febInvalidCallUpdownPatternNo(CLK:= bCallPB AND bInvalidCallUpdownPatternNoHold  , Q=> );

IF febInvalidCallUpdownPatternNo.Q THEN
bInvalidCallUpdownPatternNoPulse := TRUE;
END_IF

tInvalidCallUpdownPatternNoPulseTimer(IN:=bInvalidCallUpdownPatternNoPulse , PT:=t#0.5s , Q=> , ET=> );

IF tInvalidCallUpdownPatternNoPulseTimer.Q OR NOT bCallPB THEN
bInvalidCallUpdownPatternNoPulse := FALSE;
END_IF

IF bCallPBRE.Q AND NOT bInvalidCallUpdownPatternNoHold THEN
bCallCompleted := FALSE;
CallStep:= 1;
END_IF


CASE CallStep OF

1:

Call_DSUpdownPattern := ARDsUpdownPatternMemory[Call_iUpDownPatternNo];

CallStep := 11;


10:
bCallCompleted := TRUE;
CallSelfCheckHR := FALSE;
PreviousUpdownPatternCallNo := Call_iUpDownPatternNo;
CallStep := 99;

11:

bCallCompleted := TRUE;
CallStep := 99;



99:
;
END_CASE

END_FUNCTION_BLOCK

// ---- FBs/B_JKS_NewFB/FBP-Memory_Sub/fbA31_ArmSpeedProfileMemory.TcPOU
FUNCTION_BLOCK fbA31_ArmSpeedProfileMemory

VAR_INPUT
	bSavePB : BOOL;
	bLoadPB : BOOL;
	bCopyPB : BOOL;
	iCopyToSpdProfileNo : INT;
	iVertMaxVelo : INT;
	iVertMaxAcc : INT;
	iVertMaxDcc : INT;
	iVertMinVelo : INT;
	iVertMinAcc : INT;
	iVertMinDcc : INT;
END_VAR


VAR_IN_OUT PERSISTENT

	iArmSpdProfileNo: INT; (* 10 sets of Station Sequence Recipe *)
	DSArmSpeedProfile : DSA31_ArmSpeedProfileMemory;

	Call_iArmSpdProfile : INT;
	bCallPB: BOOL;

END_VAR
VAR_OUTPUT
	bSaveInd: BOOL;
	bLoadInd: BOOL;
	bCallCompleted : BOOL;
	bInvalidCallArmSpdProfileNoHold: BOOL;
	bInvalidCallArmSpdProfileNoPulse: BOOL;
	Call_DSArmSpeedProfile : DSA31_ArmSpeedProfileMemory;

END_VAR
VAR
	SaveIndHr: BOOL;
	LoadIndHr: BOOL;

	SaveTimerDelay: TON;
	LoadTimerDelay: TON;
	SelfCheckTimer: TON;
	bLoadEn: BOOL;
	SelfCheckloopArmSpdProfileRecipe: BOOL;
	PreviousArmSpdProfileRecipe: INT;

	LoadDF : R_TRIG;
	LoadENDF : R_TRIG;

	SaveDF: R_TRIG;
	CallIntervalTimer: TON;
	CallIntervalDIFU: R_TRIG;

	bCallCompletedHR: BOOL;
	bCallCompletedHRRE: R_TRIG;
	CallCompletedTimer: TON;
	CallSelfCheckTimer : TON;
	CallSelfCheckloop : BOOL;

	CallSelfCheckRE: R_TRIG;
	CallStep: INT;
	CallSelfCheckHR: BOOL;
	bCallPBRE: R_TRIG;

	LoadFL: INT;
	SaveFL: INT;
	PreviousArmSpdProfileCallNo: INT;
	CallSFL: INT;
	febInvalidCallArmSpdProfileNo: F_TRIG;



	rebInvalidCallArmSpdProfileNo: R_TRIG;
	tInvalidCallArmSpdProfileNoPulseTimer: TON;
	CopyDF: R_TRIG;
	iMaxMinFL: INT;
END_VAR

VAR PERSISTENT

	ARDsArmSpeedProfileMemory : ARRAY [1..iArmSpeedProfileArrayQty] OF DSA31_ArmSpeedProfileMemory;
	ARsStorageArmSpeedProfileDescription: ARRAY [0..iArmSpeedProfileArrayQty] OF STRING(50);


END_VAR

IF iArmSpdProfileNo < 1 THEN
iArmSpdProfileNo := 1;
END_IF

IF iArmSpdProfileNo > iArmSpeedProfileArrayQty THEN
iArmSpdProfileNo := iArmSpeedProfileArrayQty;
END_IF



(*Min / Max Control*)
			IF DSArmSpeedProfile.lrSpeedVelo < iVertMinVelo THEN
			DSArmSpeedProfile.lrSpeedVelo:= iVertMinVelo;
			ELSIF DSArmSpeedProfile.lrSpeedVelo > iVertMaxVelo THEN
			DSArmSpeedProfile.lrSpeedVelo:= iVertMaxVelo;
			END_IF

			IF DSArmSpeedProfile.lrAcc < iVertMinAcc THEN
			DSArmSpeedProfile.lrAcc:= iVertMinAcc;
			ELSIF DSArmSpeedProfile.lrAcc > iVertMaxAcc THEN
			DSArmSpeedProfile.lrAcc:= iVertMaxAcc;
			END_IF

			IF DSArmSpeedProfile.lrDcc < iVertMinDcc THEN
			DSArmSpeedProfile.lrDcc:= iVertMinDcc;
			ELSIF DSArmSpeedProfile.lrDcc > iVertMaxDcc THEN
			DSArmSpeedProfile.lrDcc:= iVertMaxDcc;
			END_IF



(*Load and Save Indicator*)
IF bSavePB THEN
SaveIndHr := TRUE;
END_IF

SaveTimerDelay(IN:=SaveIndHr, PT := T#1s, Q=>, ET=>);
IF SaveTimerDelay.Q THEN
SaveIndHr := FALSE;
END_IF

IF SaveIndHr AND NOT SaveTimerDelay.Q THEN
bSaveInd := TRUE;
ELSE
bSaveInd := FALSE;
END_IF

IF bLoadPB THEN
LoadIndHr := TRUE;
END_IF

LoadTimerDelay(IN:=LoadIndHr, PT := T#1s, Q=>, ET=>);
IF loadtimerdelay.Q THEN
LoadIndHr := FALSE;
END_IF

IF loadIndHr AND NOT LoadTimerDelay.Q THEN
bLoadInd := TRUE;
ELSE
bLoadInd := FALSE;
END_IF

IF iArmSpdProfileNo <> PreviousArmSpdProfileRecipe THEN
bLoadEn := TRUE;
ELSE
bLoadEn := FALSE;
END_IF


(* Load Recipe *)

LoadDF(CLK:=bLoadPB,Q=>);
LoadENDF(CLK:=bLoadEn,Q=>);

IF LoadDF.Q OR LoadENDF.Q THEN

DSArmSpeedProfile := ARDsArmSpeedProfileMemory[iArmSpdProfileNo];
PreviousArmSpdProfileRecipe := iArmSpdProfileNo  ;

END_IF


(* Save Recipe *)

SaveDF(CLK:=bSavePB,Q=>);

IF SaveDF.Q THEN

ARDsArmSpeedProfileMemory[iArmSpdProfileNo] := DSArmSpeedProfile;
ARsStorageArmSpeedProfileDescription[iArmSpdProfileNo] := DSArmSpeedProfile.sDescription;

END_IF


(*Copy Recipe*)

CopyDF(CLK:=bCopyPB,Q=>);

IF CopyDF.Q THEN

ARDsArmSpeedProfileMemory[iCopyToSpdProfileNo] := ARDsArmSpeedProfileMemory[iArmSpdProfileNo];
ARsStorageArmSpeedProfileDescription[iCopyToSpdProfileNo] := ARDsArmSpeedProfileMemory[iArmSpdProfileNo].sDescription;

END_IF





(* Call Recipe *)
(* ---- Call Recipe Complete Flag ---*)


IF NOT bCallPB THEN
bCallCompleted := FALSE;
END_IF

bCallPBRE(CLK:=bCallPB , Q=> );

IF (Call_iArmSpdProfile <= 0 OR Call_iArmSpdProfile > iArmSpeedProfileArrayQty) AND bCallPB THEN
bInvalidCallArmSpdProfileNoHold := TRUE;
ELSE
bInvalidCallArmSpdProfileNoHold := FALSE;
END_IF


febInvalidCallArmSpdProfileNo(CLK:= bCallPB AND bInvalidCallArmSpdProfileNoHold  , Q=> );

IF febInvalidCallArmSpdProfileNo.Q THEN
bInvalidCallArmSpdProfileNoPulse := TRUE;
END_IF

tInvalidCallArmSpdProfileNoPulseTimer(IN:=bInvalidCallArmSpdProfileNoPulse , PT:=t#0.5s , Q=> , ET=> );

IF tInvalidCallArmSpdProfileNoPulseTimer.Q OR NOT bCallPB THEN
bInvalidCallArmSpdProfileNoPulse := FALSE;
END_IF

IF bCallPBRE.Q AND NOT bInvalidCallArmSpdProfileNoHold THEN
bCallCompleted := FALSE;
CallStep:= 1;
END_IF


CASE CallStep OF

1:

Call_DSArmSpeedProfile := ARDsArmSpeedProfileMemory[Call_iArmSpdProfile];

CallStep := 11;


10:
bCallCompleted := TRUE;
CallSelfCheckHR := FALSE;
PreviousArmSpdProfileCallNo := Call_iArmSpdProfile;
CallStep := 99;

11:

bCallCompleted := TRUE;
CallStep := 99;



99:
;
END_CASE

END_FUNCTION_BLOCK

// ---- FBs/B_JKS_NewFB_V2/FBP-Memory_Sub/fbV2_A32_MachineZoneHeight.TcPOU
FUNCTION_BLOCK fbV2_A32_MachineZoneHeight

VAR_IN_OUT PERSISTENT

	ARDSLdZoneHeight : ARRAY [0..iLdStnQty] OF DSA32_StationZoneHeight;
	ARDSStationZoneHeight : ARRAY [0..iStnQty] OF DSA32_StationZoneHeight;
	ARDSUldZoneHeight : ARRAY [0..iUldStnQty] OF DSA32_StationZoneHeight;


END_VAR
VAR_OUTPUT
	ARDSLdZonePosOut : ARRAY [0..iLdStnQty] OF DSA32_StationZonePosOut;
	ARDSStationZonePosOut : ARRAY [0..iStnQty] OF DSA32_StationZonePosOut;
	ARDSUldZonePosOut : ARRAY [0..iUldStnQty] OF DSA32_StationZonePosOut;

END_VAR
VAR PERSISTENT

	ARfbLdStationZoneHeight : ARRAY [0..iLdStnQty] OF fbA32_StationZoneHeight;
	ARfbStationZoneHeight : ARRAY [0..iStnQty] OF fbA32_StationZoneHeight;
	ARfbUldStationZoneHeight : ARRAY [0..iUldStnQty] OF fbA32_StationZoneHeight;

END_VAR
VAR
	Loop: INT;
END_VAR

(*Loading*)

Loop := 1;
IF Loop >= 1 THEN
	FOR Loop := 1 TO iLdStnQty DO
		(*Loading*)
		IF Loop >= 1 AND Loop <= iLdStnQty THEN
		ARfbLdStationZoneHeight[Loop](DSStationZoneHeight:=ARDSLdZoneHeight[Loop] , DSStationZonePosOut=>ARDSLdZonePosOut[Loop] );
		END_IF
	END_FOR
END_IF

Loop := 1;
IF Loop >= 1 THEN
	FOR Loop := 1 TO iStnQty DO
		(*Station Qty*)
		IF Loop >= 1 AND Loop <= iStnQty THEN
		ARfbStationZoneHeight[Loop](DSStationZoneHeight:=ARDSStationZoneHeight[Loop] , DSStationZonePosOut=>ARDSStationZonePosOut[Loop] );
		END_IF
	END_FOR
END_IF

Loop := 1;
IF Loop >= 1 THEN
	FOR Loop := 1 TO iUldStnQty DO
		(*Unloading*)
		IF Loop >= 1 AND Loop <= iUldStnQty THEN
		ARfbUldStationZoneHeight[Loop](DSStationZoneHeight:=ARDSUldZoneHeight[Loop] , DSStationZonePosOut=>ARDSUldZonePosOut[Loop] );
		END_IF
	END_FOR
END_IF

END_FUNCTION_BLOCK

// ---- FBs/B_JKS_NewFB/FBP-Memory_Sub/fbA32_StationZoneHeight.TcPOU
FUNCTION_BLOCK fbA32_StationZoneHeight
VAR_IN_OUT PERSISTENT

	DSStationZoneHeight : DSA32_StationZoneHeight;


END_VAR
VAR_OUTPUT
	DSStationZonePosOut : DSA32_StationZonePosOut;

END_VAR
VAR
	bZone1RangeValid: BOOL;
	bZone2RangeValid: BOOL;
	bZone3RangeValid: BOOL;
	bZone4RangeValid: BOOL;
END_VAR

DSStationZonePosOut.lrZone1StartPos := DSStationZoneHeight.lrTopPos;
DSStationZonePosOut.lrZone2StartPos := DSStationZonePosOut.lrZone1EndPos;
DSStationZonePosOut.lrZone3StartPos := DSStationZonePosOut.lrZone2EndPos;
DSStationZonePosOut.lrZone4StartPos := DSStationZonePosOut.lrZone3EndPos;

DSStationZonePosOut.lrZone1EndPos := DSStationZoneHeight.lrTopPos + DSStationZoneHeight.lrZone1Range;
DSStationZonePosOut.lrZone2EndPos := DSStationZoneHeight.lrTopPos + DSStationZoneHeight.lrZone1Range + DSStationZoneHeight.lrZone2Range;
DSStationZonePosOut.lrZone3EndPos := DSStationZoneHeight.lrTopPos + DSStationZoneHeight.lrZone1Range + DSStationZoneHeight.lrZone2Range + DSStationZoneHeight.lrZone3Range;
DSStationZonePosOut.lrZone4EndPos := DSStationZoneHeight.lrBottomPos;

DSStationZonePosOut.lrMidPos := DSStationZoneHeight.lrMidPos; (*Added New*)

DSStationZoneHeight.lrZone4Range := DSStationZoneHeight.lrBottomPos - DSStationZonePosOut.lrZone3EndPos;

IF DSStationZoneHeight.lrZone1Range > (DSStationZoneHeight.lrBottomPos - DSStationZoneHeight.lrTopPos) THEN
DSStationZoneHeight.lrZone1Range := DSStationZoneHeight.lrBottomPos - DSStationZoneHeight.lrTopPos;
END_IF

IF DSStationZoneHeight.lrZone2Range > (DSStationZoneHeight.lrBottomPos - DSStationZoneHeight.lrZone1Range - DSStationZoneHeight.lrTopPos) THEN
DSStationZoneHeight.lrZone2Range := DSStationZoneHeight.lrBottomPos - DSStationZoneHeight.lrZone1Range - DSStationZoneHeight.lrTopPos;
END_IF

IF DSStationZoneHeight.lrZone3Range > (DSStationZoneHeight.lrBottomPos - DSStationZoneHeight.lrZone1Range - DSStationZoneHeight.lrZone2Range - DSStationZoneHeight.lrTopPos) THEN
DSStationZoneHeight.lrZone3Range := DSStationZoneHeight.lrBottomPos - DSStationZoneHeight.lrZone1Range - DSStationZoneHeight.lrZone2Range - DSStationZoneHeight.lrTopPos;
END_IF


IF DSStationZoneHeight.lrZone1Range < 0 THEN
DSStationZoneHeight.lrZone1Range := 0;
ELSIF DSStationZoneHeight.lrZone2Range < 0 THEN
DSStationZoneHeight.lrZone2Range := 0;
ELSIF DSStationZoneHeight.lrZone3Range < 0 THEN
DSStationZoneHeight.lrZone3Range := 0;
END_IF







IF DSStationZoneHeight.lrZone1Range <> 0 THEN
bZone1RangeValid := TRUE;
ELSE
bZone1RangeValid := FALSE;
END_IF

IF DSStationZoneHeight.lrZone2Range <> 0 THEN
bZone2RangeValid := TRUE;
ELSE
bZone2RangeValid := FALSE;
END_IF

IF DSStationZoneHeight.lrZone3Range <> 0 THEN
bZone3RangeValid := TRUE;
ELSE
bZone3RangeValid := FALSE;
END_IF

IF DSStationZoneHeight.lrZone4Range <> 0 THEN
bZone4RangeValid := TRUE;
ELSE
bZone4RangeValid := FALSE;
END_IF

END_FUNCTION_BLOCK

// ---- POUs/MainProgram/AutoArmCtrl/PosConfirmBitCtrl_Arm1.TcPOU
PROGRAM PosConfirmBitCtrl_Arm1
VAR

	fbFBPArmHorzZoneConfirm_Arm1 : fbV2_FBPArmHorzZoneConfirm;

END_VAR

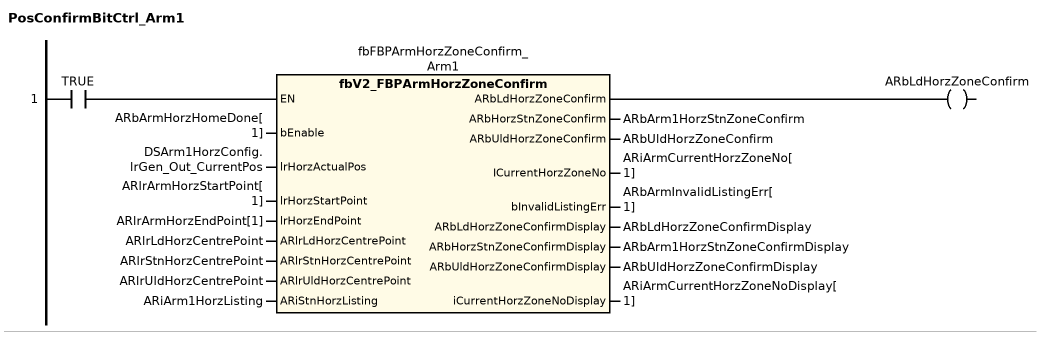
// NETWORK 1
fbFBPArmHorzZoneConfirm_Arm1(
    bEnable := ARbArmHorzHomeDone[1],
    lrHorzActualPos := DSArm1HorzConfig.lrGen_Out_CurrentPos,
    lrHorzStartPoint := ARlrArmHorzStartPoint[1],
    lrHorzEndPoint := ARlrArmHorzEndPoint[1],
    ARlrLdHorzCentrePoint := ARlrLdHorzCentrePoint,
    ARlrStnHorzCentrePoint := ARlrStnHorzCentrePoint,
    ARlrUldHorzCentrePoint := ARlrUldHorzCentrePoint,
    ARiStnHorzListing := ARiArm1HorzListing,
    ARbHorzStnZoneConfirm => ARbArm1HorzStnZoneConfirm,
    ARbUldHorzZoneConfirm => ARbUldHorzZoneConfirm,
    ICurrentHorzZoneNo => ARiArmCurrentHorzZoneNo[1],
    bInvalidListingErr => ARbArmInvalidListingErr[1],
    ARbLdHorzZoneConfirmDisplay => ARbLdHorzZoneConfirmDisplay,
    ARbHorzStnZoneConfirmDisplay => ARbArm1HorzStnZoneConfirmDisplay,
    ARbUldHorzZoneConfirmDisplay => ARbUldHorzZoneConfirmDisplay,
    iCurrentHorzZoneNoDisplay => ARiArmCurrentHorzZoneNoDisplay[1]); // fbV2_FBPArmHorzZoneConfirm
ARbLdHorzZoneConfirm := fbFBPArmHorzZoneConfirm_Arm1.ARbLdHorzZoneConfirm;

END_PROGRAM

// ---- FBs/B_JKS_NewFB_V2/FBP-ArmRelated/fbV2_FBPArmHorzZoneConfirm.TcPOU
FUNCTION_BLOCK fbV2_FBPArmHorzZoneConfirm
VAR_INPUT
	bEnable 					: BOOL;
(*	ARiLdStnID					: INT;
	ARiUldStnID					: INT;
*)	lrHorzActualPos 			: LREAL;
	lrHorzStartPoint 			: LREAL;
	lrHorzEndPoint 			: LREAL;
	ARlrLdHorzCentrePoint 	: ARRAY [0..iLdStnQty] OF LREAL;
	ARlrStnHorzCentrePoint 	: ARRAY [0..iStnQty] OF LREAL;
	ARlrUldHorzCentrePoint 	: ARRAY [0..iUldStnQty] OF LREAL;
	ARiStnHorzListing 		: ARRAY [1..50] OF INT;

END_VAR


VAR_OUTPUT
	ARbLdHorzZoneConfirm 		: ARRAY [0..iLdStnQty] OF BOOL;
	ARbHorzStnZoneConfirm 		: ARRAY [1..iStnQty] OF BOOL;
	ARbUldHorzZoneConfirm 		: ARRAY [0..iUldStnQty] OF BOOL;
	ICurrentHorzZoneNo 			: INT;
	bInvalidListingErr				: BOOL;

	ARbLdHorzZoneConfirmDisplay 		: ARRAY [0..iLdStnQty] OF BOOL;
	ARbHorzStnZoneConfirmDisplay 	: ARRAY [1..iStnQty] OF BOOL;
	ARbUldHorzZoneConfirmDisplay 	: ARRAY [0..iUldStnQty] OF BOOL;
	iCurrentHorzZoneNoDisplay 		: INT;

END_VAR
(*
VAR_IN_OUT
	iZoneEndPoint : ARRAY [1..20] OF INT;
	iActualPos: INT;

END_VAR
*)
VAR

	iActualPos: INT;


	bEnableRE: R_TRIG;
	iGenZoneFL: INT;
	ARlrZoneCentrePoint : ARRAY [1..50] OF LREAL;
	ARlrZoneEndPoint : ARRAY [1..50] OF LREAL;
	ARbZonePosConfirmInt : ARRAY [1..50] OF BOOL;
	iCheckListFL: INT;
	iEndPointFL: INT;
	bEnableFE: F_TRIG;
	iClearFL: INT;
	IZonePosCfFL: INT;
	iCurrentStnFL: INT;
	bCheckStnConfirm: BOOL;
	iCheckStnBitFL: INT;
	iGenZoneSFL: INT;
	bStnHorzListingFound: BOOL;
	bCurrentHorzZoneNoFound: BOOL;
END_VAR

(*bEnable Rising Edge*)
bEnableRE(CLK:=bEnable , Q=> );
bEnableFE(CLK:=bEnable , Q=> );


(*Generate Zone Centre Point and Transfer Confirm Bit*)
IF bEnable THEN
iGenZoneFL := 1;
	FOR iGenZoneFL := 1 TO 50 DO
		IF iGenZoneFL >= 1 AND iGenZoneFL <= 50 THEN

		bStnHorzListingFound := FALSE;

			iGenZoneSFL := 1;
				FOR iGenZoneSFL := 1 TO iLdStnQty DO
					IF iGenZoneSFL >= 1 AND iGenZoneSFL <= iLdStnQty THEN

						IF ARiStnHorzListing[iGenZoneFL] = ARiLdStnID[iGenZoneSFL] THEN
							ARlrZoneCentrePoint[iGenZoneFL] := ARlrLdHorzCentrePoint[iGenZoneSFL];
							ARbLdHorzZoneConfirm[iGenZoneSFL] := ARbZonePosConfirmInt[iGenZoneFL];
							bStnHorzListingFound := TRUE;
						END_IF

					END_IF
				END_FOR

			iGenZoneSFL := 1;
				FOR iGenZoneSFL := 1 TO iUldStnQty DO
					IF iGenZoneSFL >= 1 AND iGenZoneSFL <= iUldStnQty THEN

						IF ARiStnHorzListing[iGenZoneFL] = ARiUldStnID[iGenZoneSFL] THEN
							ARlrZoneCentrePoint[iGenZoneFL] := ARlrUldHorzCentrePoint[iGenZoneSFL];
							ARbUldHorzZoneConfirm[iGenZoneSFL] := ARbZonePosConfirmInt[iGenZoneFL];
							bStnHorzListingFound := TRUE;
						END_IF

					END_IF
				END_FOR


			IF NOT bStnHorzListingFound (*ARiStnHorzListing[iGenZoneFL] <> ARiUldStnID AND ARiStnHorzListing[iGenZoneFL] <> ARiUldStnID*) AND ARiStnHorzListing[iGenZoneFL] <> 0 AND ARiStnHorzListing[iGenZoneFL] <= iStnQty THEN
				ARlrZoneCentrePoint[iGenZoneFL] := ARlrStnHorzCentrePoint[ARiStnHorzListing[iGenZoneFL]];
				ARbHorzStnZoneConfirm[ARiStnHorzListing[iGenZoneFL]] := ARbZonePosConfirmInt[iGenZoneFL];
			END_IF


		END_IF
	END_FOR
END_IF


(*Check invalid Stn Listing*)
IF bEnableRE.Q THEN
bInvalidListingErr := FALSE;
iCheckListFL := 1;
	FOR iCheckListFL := 1 TO 50 DO
		IF iCheckListFL >= 1 AND iCheckListFL <= 50 THEN

			IF iCheckListFL = 1 AND ARlrZoneCentrePoint[1] <= 0 THEN
			bInvalidListingErr := TRUE;
			iCheckListFL := 50+1;
			END_IF

			IF iCheckListFL > 1 AND ARlrZoneCentrePoint[iCheckListFL] <= ARlrZoneCentrePoint[iCheckListFL-1] AND ARiStnHorzListing[iCheckListFL] >0 THEN
			bInvalidListingErr := TRUE;
			iCheckListFL := 50+1;
			END_IF
		END_IF
	END_FOR
END_IF




(*Generate End Point *)
IF bEnableRE.Q THEN
iEndPointFL := 1;
	FOR iEndPointFL := 1 TO 50 DO
		IF iEndPointFL >= 1 AND iEndPointFL <= 50-1 THEN

(*			IF iEndPointFL >1 THEN*)
				IF ((ARlrZoneCentrePoint[iEndPointFL+1] - ARlrZoneCentrePoint[iEndPointFL])/2) >0 THEN
				ARlrZoneEndPoint[iEndPointFL] := ((ARlrZoneCentrePoint[iEndPointFL+1] - ARlrZoneCentrePoint[iEndPointFL])/2)+ARlrZoneCentrePoint[iEndPointFL];
				ELSIF lrHorzEndPoint <= ARlrZoneCentrePoint[iEndPointFL] THEN
				ARlrZoneEndPoint[iEndPointFL] := ARlrZoneCentrePoint[iEndPointFL]+5000;
				iEndPointFL := 50+1;
				ELSIF lrHorzEndPoint > ARlrZoneCentrePoint[iEndPointFL] THEN
				ARlrZoneEndPoint[iEndPointFL] := lrHorzEndPoint+1;
				iEndPointFL := 50+1;
				END_IF
(*			END_IF*)
		END_IF
	END_FOR
END_IF


(*Clear Data*)
IF bEnableFE.Q THEN
iClearFL := 1;
	FOR iClearFL := 1 TO 50 DO
		IF iClearFL >= 1 AND iClearFL <= 50 THEN

			ARlrZoneCentrePoint[iClearFL] := 0;
			ARlrZoneEndPoint[iClearFL] := 0;
			ARbZonePosConfirmInt[iClearFL] := FALSE;

			IF iClearFL >= 1 AND iClearFL <= iStnQty THEN
			ARbHorzStnZoneConfirm[iClearFL] := FALSE;
			END_IF

			IF iClearFL >= 1 AND iClearFL <= iLdStnQty THEN
			ARbLdHorzZoneConfirm[iClearFL] := FALSE;
			END_IF

			IF iClearFL >= 1 AND iClearFL <= iUldStnQty THEN
			ARbUldHorzZoneConfirm[iClearFL] := FALSE;
			END_IF

		END_IF
	END_FOR



ICurrentHorzZoneNo := 0;
bInvalidListingErr := FALSE;
END_IF


(*Convert LREAL to INT*)


iActualPos := LREAL_TO_INT(lrHorzActualPos);




IF bEnable AND NOT bInvalidListingErr THEN


(*General Zone Pos Confirm Internal*)
IZonePosCfFL := 1;
	FOR IZonePosCfFL := 1 TO 50 DO
		IF IZonePosCfFL >= 1 AND IZonePosCfFL <= 50 THEN

			IF IZonePosCfFL = 1 THEN
				IF (iActualPos >= lrHorzStartPoint) AND (iActualPos < ARlrZoneEndPoint[IZonePosCfFL]) AND iActualPos >0 THEN
				ARbZonePosConfirmInt[IZonePosCfFL] := TRUE;
				ELSE
				ARbZonePosConfirmInt[IZonePosCfFL] := FALSE;
				END_IF
			END_IF

			IF IZonePosCfFL > 1 THEN
				IF (iActualPos >= ARlrZoneEndPoint[IZonePosCfFL-1]) AND (iActualPos < ARlrZoneEndPoint[IZonePosCfFL]) AND iActualPos >0 THEN
				ARbZonePosConfirmInt[IZonePosCfFL] := TRUE;
				ELSE
				ARbZonePosConfirmInt[IZonePosCfFL] := FALSE;
				END_IF
			END_IF
		END_IF
	END_FOR

(*Generate ICurrentHorzZoneNo *)
	bCurrentHorzZoneNoFound := FALSE;


		IF NOT bCurrentHorzZoneNoFound THEN

		iCurrentStnFL := 1;
			FOR iCurrentStnFL := 1 TO iLdStnQty DO
				IF iCurrentStnFL >= 1 AND iCurrentStnFL <= iLdStnQty THEN

					IF ARbLdHorzZoneConfirm[iCurrentStnFL] THEN
					ICurrentHorzZoneNo := ARiLdStnID[iCurrentStnFL];
					bCurrentHorzZoneNoFound := TRUE;
					END_IF

				END_IF
			END_FOR
		END_IF


		IF NOT bCurrentHorzZoneNoFound THEN

		iCurrentStnFL := 1;
			FOR iCurrentStnFL := 1 TO iUldStnQty DO
				IF iCurrentStnFL >= 1 AND iCurrentStnFL <= iUldStnQty THEN

					IF ARbUldHorzZoneConfirm[iCurrentStnFL] THEN
					ICurrentHorzZoneNo := ARiUldStnID[iCurrentStnFL];
					bCurrentHorzZoneNoFound := TRUE;
					END_IF

				END_IF
			END_FOR
		END_IF

		IF NOT bCurrentHorzZoneNoFound THEN

		iCurrentStnFL := 1;
			FOR iCurrentStnFL := 1 TO iStnQty DO
				IF iCurrentStnFL >= 1 AND iCurrentStnFL <= iStnQty THEN

					IF ARbHorzStnZoneConfirm[iCurrentStnFL] THEN
					ICurrentHorzZoneNo := iCurrentStnFL;
					bCurrentHorzZoneNoFound := TRUE;
					END_IF

				END_IF
			END_FOR
		END_IF
(*
(*Check if any Ld/Uld/Stn Pos Confirm Bit is on, else -> ICurrentHorzZoneNo := 0; *)
bCheckStnConfirm := FALSE;
iCheckStnBitFL := 1;

	FOR iCheckStnBitFL := 1 TO iStnQty DO
		IF iCheckStnBitFL >= 1 AND iCheckStnBitFL <= iStnQty THEN
			IF ARbHorzStnZoneConfirm[iCheckStnBitFL] THEN
			bCheckStnConfirm := TRUE;
			END_IF
		END_IF
	END_FOR

*)
	IF NOT bCurrentHorzZoneNoFound(*ARbLdHorzZoneConfirm AND NOT ARbUldHorzZoneConfirm AND NOT bCheckStnConfirm*) THEN
	ICurrentHorzZoneNo := 0;
	END_IF

END_IF



(*Edit by Lee - Generate the Position Confirm Signal (Just Display) even though the Arm is no HOMING - 20180119*)
(*Generate Zone Centre Point and Transfer Confirm Bit*)
IF NOT bEnable THEN
iGenZoneFL := 1;
	FOR iGenZoneFL := 1 TO 50 DO
		IF iGenZoneFL >= 1 AND iGenZoneFL <= 50 THEN

		bStnHorzListingFound := FALSE;

			iGenZoneSFL := 1;
				FOR iGenZoneSFL := 1 TO iLdStnQty DO
					IF iGenZoneSFL >= 1 AND iGenZoneSFL <= iLdStnQty THEN

						IF ARiStnHorzListing[iGenZoneFL] = ARiLdStnID[iGenZoneSFL] THEN
							ARlrZoneCentrePoint[iGenZoneFL] := ARlrLdHorzCentrePoint[iGenZoneSFL];
							ARbLdHorzZoneConfirmDisplay[iGenZoneSFL] := ARbZonePosConfirmInt[iGenZoneFL];
							bStnHorzListingFound := TRUE;
						END_IF

					END_IF
				END_FOR

			iGenZoneSFL := 1;
				FOR iGenZoneSFL := 1 TO iUldStnQty DO
					IF iGenZoneSFL >= 1 AND iGenZoneSFL <= iUldStnQty THEN

						IF ARiStnHorzListing[iGenZoneFL] = ARiUldStnID[iGenZoneSFL] THEN
							ARlrZoneCentrePoint[iGenZoneFL] := ARlrUldHorzCentrePoint[iGenZoneSFL];
							ARbUldHorzZoneConfirmDisplay[iGenZoneSFL] := ARbZonePosConfirmInt[iGenZoneFL];
							bStnHorzListingFound := TRUE;
						END_IF

					END_IF
				END_FOR


			IF NOT bStnHorzListingFound (*ARiStnHorzListing[iGenZoneFL] <> ARiUldStnID AND ARiStnHorzListing[iGenZoneFL] <> ARiUldStnID*) AND ARiStnHorzListing[iGenZoneFL] <> 0 AND ARiStnHorzListing[iGenZoneFL] <= iStnQty THEN
				ARlrZoneCentrePoint[iGenZoneFL] := ARlrStnHorzCentrePoint[ARiStnHorzListing[iGenZoneFL]];
				ARbHorzStnZoneConfirmDisplay[ARiStnHorzListing[iGenZoneFL]] := ARbZonePosConfirmInt[iGenZoneFL];
			END_IF

		END_IF
	END_FOR
END_IF

(*Edit by Lee - Generate the Position Confirm Signal (Just Display) even though the Arm is no HOMING - 20180119*)
(*Generate End Point *)
IF NOT bEnable THEN
iEndPointFL := 1;
	FOR iEndPointFL := 1 TO 50 DO
		IF iEndPointFL >= 1 AND iEndPointFL <= 50-1 THEN

(*			IF iEndPointFL >1 THEN*)
				IF ((ARlrZoneCentrePoint[iEndPointFL+1] - ARlrZoneCentrePoint[iEndPointFL])/2) >0 THEN
				ARlrZoneEndPoint[iEndPointFL] := ((ARlrZoneCentrePoint[iEndPointFL+1] - ARlrZoneCentrePoint[iEndPointFL])/2)+ARlrZoneCentrePoint[iEndPointFL];
				ELSIF lrHorzEndPoint <= ARlrZoneCentrePoint[iEndPointFL] THEN
				ARlrZoneEndPoint[iEndPointFL] := ARlrZoneCentrePoint[iEndPointFL]+5000;
				iEndPointFL := 50+1;
				ELSIF lrHorzEndPoint > ARlrZoneCentrePoint[iEndPointFL] THEN
				ARlrZoneEndPoint[iEndPointFL] := lrHorzEndPoint+1;
				iEndPointFL := 50+1;
				END_IF
(*			END_IF*)
		END_IF
	END_FOR
END_IF


IF NOT bEnable AND NOT bInvalidListingErr THEN

(*Edit by Lee - Generate the Position Confirm Signal (Just Display) even though the Arm is no HOMING - 20180119*)
(*General Zone Pos Confirm Internal*)
IZonePosCfFL := 1;
	FOR IZonePosCfFL := 1 TO 50 DO
		IF IZonePosCfFL >= 1 AND IZonePosCfFL <= 50 THEN

			IF IZonePosCfFL = 1 THEN
				IF (iActualPos >= lrHorzStartPoint) AND (iActualPos < ARlrZoneEndPoint[IZonePosCfFL]) AND iActualPos >0 THEN
				ARbZonePosConfirmInt[IZonePosCfFL] := TRUE;
				ELSE
				ARbZonePosConfirmInt[IZonePosCfFL] := FALSE;
				END_IF
			END_IF

			IF IZonePosCfFL > 1 THEN
				IF (iActualPos >= ARlrZoneEndPoint[IZonePosCfFL-1]) AND (iActualPos < ARlrZoneEndPoint[IZonePosCfFL]) AND iActualPos >0 THEN
				ARbZonePosConfirmInt[IZonePosCfFL] := TRUE;
				ELSE
				ARbZonePosConfirmInt[IZonePosCfFL] := FALSE;
				END_IF
			END_IF
		END_IF
	END_FOR

(*Edit by Lee - Generate the Position Confirm Signal (Just Display) even though the Arm is no HOMING - 20180119*)
(*Generate ICurrentHorzZoneNo *)
	bCurrentHorzZoneNoFound := FALSE;


		IF NOT bCurrentHorzZoneNoFound THEN

		iCurrentStnFL := 1;
			FOR iCurrentStnFL := 1 TO iLdStnQty DO
				IF iCurrentStnFL >= 1 AND iCurrentStnFL <= iLdStnQty THEN

					IF ARbLdHorzZoneConfirmDisplay[iCurrentStnFL] THEN
					iCurrentHorzZoneNoDisplay := ARiLdStnID[iCurrentStnFL];
					bCurrentHorzZoneNoFound := TRUE;
					END_IF

				END_IF
			END_FOR
		END_IF


		IF NOT bCurrentHorzZoneNoFound THEN

		iCurrentStnFL := 1;
			FOR iCurrentStnFL := 1 TO iUldStnQty DO
				IF iCurrentStnFL >= 1 AND iCurrentStnFL <= iUldStnQty THEN

					IF ARbUldHorzZoneConfirmDisplay[iCurrentStnFL] THEN
					iCurrentHorzZoneNoDisplay := ARiUldStnID[iCurrentStnFL];
					bCurrentHorzZoneNoFound := TRUE;
					END_IF

				END_IF
			END_FOR
		END_IF

		IF NOT bCurrentHorzZoneNoFound THEN

		iCurrentStnFL := 1;
			FOR iCurrentStnFL := 1 TO iStnQty DO
				IF iCurrentStnFL >= 1 AND iCurrentStnFL <= iStnQty THEN

					IF ARbHorzStnZoneConfirmDisplay[iCurrentStnFL] THEN
					iCurrentHorzZoneNoDisplay := iCurrentStnFL;
					bCurrentHorzZoneNoFound := TRUE;
					END_IF

				END_IF
			END_FOR
		END_IF

	IF NOT bCurrentHorzZoneNoFound THEN
	iCurrentHorzZoneNoDisplay := 0;
	END_IF

END_IF

END_FUNCTION_BLOCK

// ---- POUs/MainProgram/Barcode/BarcodeCtrl_Utac.TcPOU

PROGRAM BarcodeCtrl_Utac
VAR
	bTestsensor:BOOL;
	(*X120_00*)

END_VAR

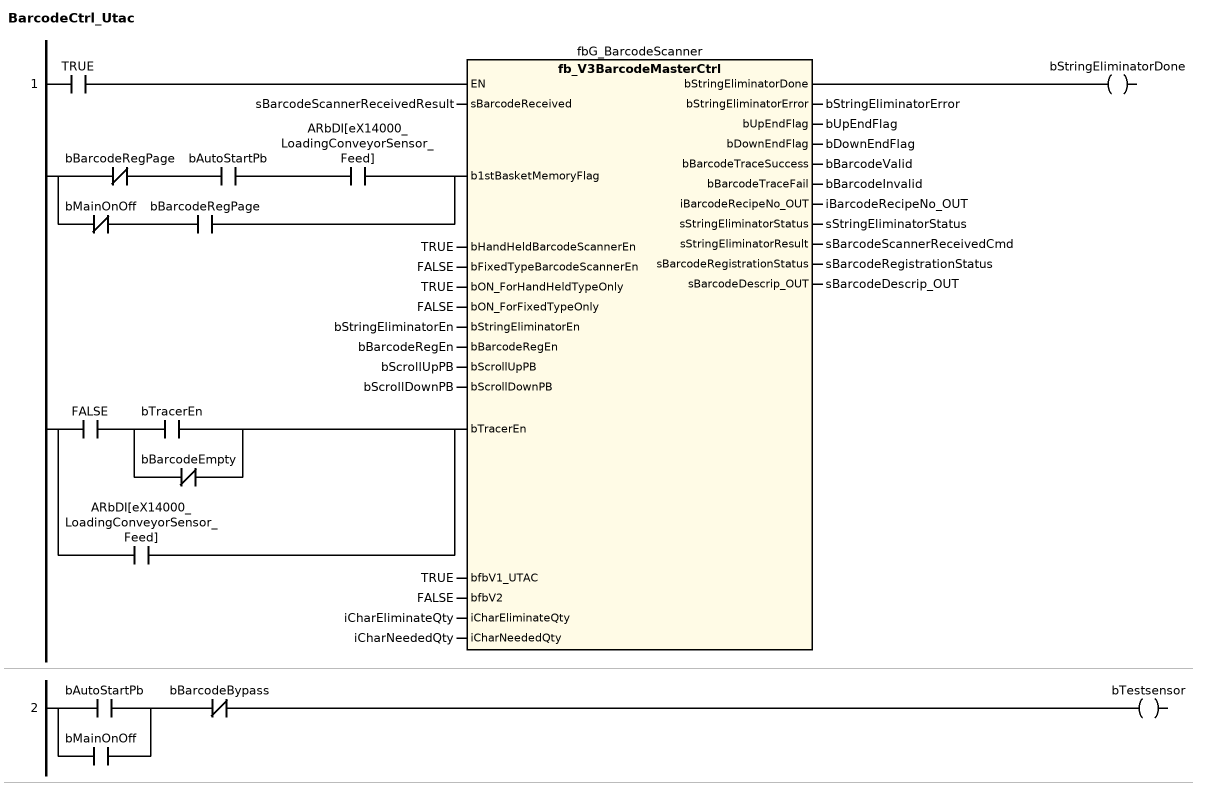
// NETWORK 1
fbG_BarcodeScanner(
    sBarcodeReceived := sBarcodeScannerReceivedResult,
    b1stBasketMemoryFlag := NOT bBarcodeRegPage AND bAutoStartPb AND ARbDI[eX14000_LoadingConveyorSensor_Feed] OR NOT bMainOnOff AND bBarcodeRegPage,
    bHandHeldBarcodeScannerEn := TRUE,
    bFixedTypeBarcodeScannerEn := FALSE,
    bON_ForHandHeldTypeOnly := TRUE,
    bON_ForFixedTypeOnly := FALSE,
    bStringEliminatorEn := bStringEliminatorEn,
    bBarcodeRegEn := bBarcodeRegEn,
    bScrollUpPB := bScrollUpPB,
    bScrollDownPB := bScrollDownPB,
    bTracerEn := FALSE AND (bTracerEn OR NOT bBarcodeEmpty) OR ARbDI[eX14000_LoadingConveyorSensor_Feed],
    bfbV1_UTAC := TRUE,
    bfbV2 := FALSE,
    iCharEliminateQty := iCharEliminateQty,
    iCharNeededQty := iCharNeededQty,
    bStringEliminatorError => bStringEliminatorError,
    bUpEndFlag => bUpEndFlag,
    bDownEndFlag => bDownEndFlag,
    bBarcodeTraceSuccess => bBarcodeValid,
    bBarcodeTraceFail => bBarcodeInvalid,
    iBarcodeRecipeNo_OUT => iBarcodeRecipeNo_OUT,
    sStringEliminatorStatus => sStringEliminatorStatus,
    sStringEliminatorResult => sBarcodeScannerReceivedCmd,
    sBarcodeRegistrationStatus => sBarcodeRegistrationStatus,
    sBarcodeDescrip_OUT => sBarcodeDescrip_OUT); // fb_V3BarcodeMasterCtrl
bStringEliminatorDone := fbG_BarcodeScanner.bStringEliminatorDone;

// NETWORK 2
bTestsensor := (bAutoStartPb OR bMainOnOff) AND NOT bBarcodeBypass;

END_PROGRAM

// ---- FBs/fbV3BarcodeCtrl/Main FB/fb_V3BarcodeMasterCtrl.TcPOU
FUNCTION_BLOCK fb_V3BarcodeMasterCtrl
VAR_INPUT
	
	sBarcodeReceived								: STRING;
	b1stBasketMemoryFlag							: BOOL;
	bHandHeldBarcodeScannerEn 						: BOOL;
	bFixedTypeBarcodeScannerEn 						: BOOL;
	bON_ForHandHeldTypeOnly 						: BOOL;
	bON_ForFixedTypeOnly 							: BOOL;
	bStringEliminatorEn 								: BOOL;
	bBarcodeRegEn 									: BOOL;
	bScrollUpPB 										: BOOL;
	bScrollDownPB 									: BOOL;
	bTracerEn 										: BOOL;
	bfbV1_UTAC 										: BOOL;
	bfbV2 											: BOOL;
	iCharEliminateQty 									: INT;
	iCharNeededQty 									: INT;
(*
	ARsBarCodeRaw_V2 : ARRAY [0..99] OF STRING;
	ARsBarcodeDescrip_V2 : ARRAY [0..99] OF STRING;
*)

END_VAR

VAR_IN_OUT
END_VAR

VAR_OUTPUT
	bStringEliminatorDone 								: BOOL;
	bStringEliminatorError								: BOOL;
	bUpEndFlag 										: BOOL;
	bDownEndFlag 									: BOOL;
	bBarcodeTraceSuccess 							: BOOL;
	bBarcodeTraceFail 								: BOOL;
	iBarcodeRecipeNo_OUT 							: INT;
	sStringEliminatorStatus 							: STRING(50);
	sStringEliminatorResult 							: STRING;
	sBarcodeRegistrationStatus 						: STRING;
	sBarcodeDescrip_OUT 							: STRING;
(*
	sSendString						: STRING;
	sReceivedString					: STRING;
*)
END_VAR
VAR
	fbV3BarcodeScanner								: fb_V3BarcodeScanner;
	fbV3StringEliminator 								: fb_V3StringEliminator;
	fbV1BarcodeRegistration 							: fb_V1BarcodeRegistration_UTAC;
	fbV2BarcodeRegistration							: fb_V2BarcodeRegistration;
	fbV3BarcodeTracer 								: fb_V3BarcodeTracer;
	fbV3BarcodeRegSectionDisplayController 			: fb_V3BarcodeRegSectionDisplayController;

	sReceivedString									: STRING;

END_VAR
VAR // added by the converter: edge detectors and wires of the graphical bodies
    _w1 : STRING(INT#0);
END_VAR

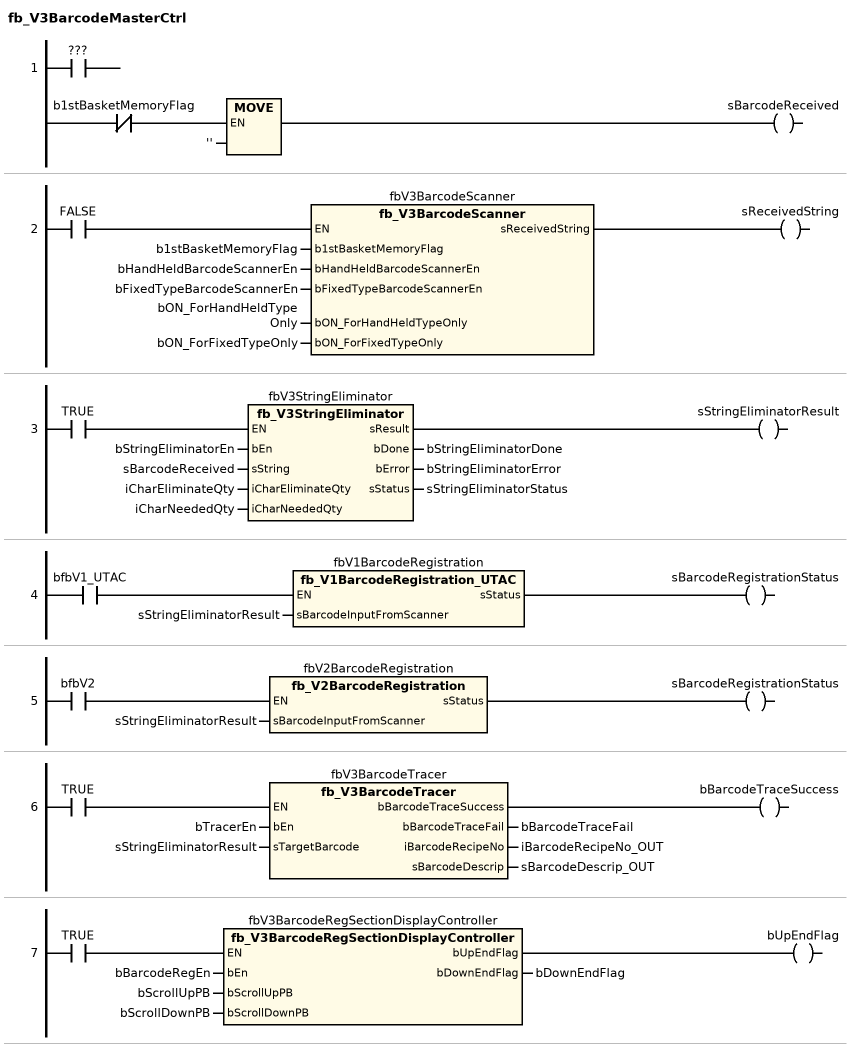
// NETWORK 1
IF NOT b1stBasketMemoryFlag THEN _w1 := ''; END_IF
sBarcodeReceived := _w1;

// NETWORK 2
IF FALSE THEN
    fbV3BarcodeScanner(
        b1stBasketMemoryFlag := b1stBasketMemoryFlag,
        bHandHeldBarcodeScannerEn := bHandHeldBarcodeScannerEn,
        bFixedTypeBarcodeScannerEn := bFixedTypeBarcodeScannerEn,
        bON_ForHandHeldTypeOnly := bON_ForHandHeldTypeOnly,
        bON_ForFixedTypeOnly := bON_ForFixedTypeOnly); // fb_V3BarcodeScanner
END_IF
sReceivedString := fbV3BarcodeScanner.sReceivedString;

// NETWORK 3
fbV3StringEliminator(
    bEn := bStringEliminatorEn,
    sString := sBarcodeReceived,
    iCharEliminateQty := iCharEliminateQty,
    iCharNeededQty := iCharNeededQty,
    bDone => bStringEliminatorDone,
    bError => bStringEliminatorError,
    sStatus => sStringEliminatorStatus); // fb_V3StringEliminator
sStringEliminatorResult := fbV3StringEliminator.sResult;

// NETWORK 4
IF bfbV1_UTAC THEN
    fbV1BarcodeRegistration(sBarcodeInputFromScanner := sStringEliminatorResult); // fb_V1BarcodeRegistration_UTAC
END_IF
sBarcodeRegistrationStatus := fbV1BarcodeRegistration.sStatus;

// NETWORK 5
IF bfbV2 THEN
    fbV2BarcodeRegistration(sBarcodeInputFromScanner := sStringEliminatorResult); // fb_V2BarcodeRegistration
END_IF
sBarcodeRegistrationStatus := fbV2BarcodeRegistration.sStatus;

// NETWORK 6
fbV3BarcodeTracer(
    bEn := bTracerEn,
    sTargetBarcode := sStringEliminatorResult,
    bBarcodeTraceFail => bBarcodeTraceFail,
    iBarcodeRecipeNo => iBarcodeRecipeNo_OUT,
    sBarcodeDescrip => sBarcodeDescrip_OUT); // fb_V3BarcodeTracer
bBarcodeTraceSuccess := fbV3BarcodeTracer.bBarcodeTraceSuccess;

// NETWORK 7
fbV3BarcodeRegSectionDisplayController(
    bEn := bBarcodeRegEn,
    bScrollUpPB := bScrollUpPB,
    bScrollDownPB := bScrollDownPB,
    bDownEndFlag => bDownEndFlag); // fb_V3BarcodeRegSectionDisplayController
bUpEndFlag := fbV3BarcodeRegSectionDisplayController.bUpEndFlag;

END_FUNCTION_BLOCK

// ---- FBs/fbV3BarcodeCtrl/Sub FB/fb_V3BarcodeScanner.TcPOU
FUNCTION_BLOCK fb_V3BarcodeScanner
VAR_INPUT
	b1stBasketMemoryFlag		: BOOL;
	bHandHeldBarcodeScannerEn : BOOL;
	bFixedTypeBarcodeScannerEn : BOOL;
	bON_ForHandHeldTypeOnly : BOOL;
	bON_ForFixedTypeOnly : BOOL;

END_VAR

VAR_OUTPUT
	sReceivedString : STRING;

END_VAR

VAR_IN_OUT
END_VAR

VAR
	bEnable  						: BOOL;
	bSendString						: BOOL;
	tOn_1s							: TON;
	tOn_Delay						: TON;
	tOff_Refresh						: TON;

	bOn							: BOOL;

	tOn_DelayRE						: R_TRIG;
	tOff_RefreshRE					: R_TRIG;

	byStep							: BYTE;

	fbReceiveString 					: ReceiveString;
	fbReceiveString_Rst				: BOOL;
	fbReceiveString_StrRcv			: BOOL;

	fbSendString255					: SendString;
	Busy							: BOOL;
	Error							: comerror_t;

	sDelimiteChar					: STRING:='$R';
	sReceivedStringRaw				: STRING;
	iReceivedStingProcess			: INT;

	(*sReceivedStringRaw2				: STRING;*)

	SerialLineControl : SerialLineControl;

	SerInDataCom		AT%I*		: EL6inData22B;
	SerOutDataCom		AT%Q*		: EL6OutData22B;
	BufferReadCom					: ComBuffer;
	BufferWriteCom					: ComBuffer;

	sSendString						: STRING;

	tReceivedString_DelayReset		: TON;
END_VAR

(* To determine whether use FixedType or Handheld Barcode Scanner*)

IF NOT bHandHeldBarcodeScannerEn AND bFixedTypeBarcodeScannerEn AND bON_ForFixedTypeOnly THEN
bON := TRUE;
ELSE
bON := FALSE;
END_IF

(*** for FixedType Scanner***)
IF NOT bHandHeldBarcodeScannerEn AND bFixedTypeBarcodeScannerEn THEN

			(*bON is "ON" --> Trigger 1 time sending*)
			
			tOn_Delay(IN:=bON, PT:=t#0.5s , Q=> , ET=> );

			tOn_DelayRE(CLK:=tOn_Delay.Q AND bON,Q=>);
			IF tOn_DelayRE.Q THEN
				byStep:= 10;
			END_IF

			(*bON is "OFF" --> Trigger always OFF reflash*)

			tOff_Refresh(IN:=NOT tOff_Refresh.Q AND NOT bON, PT:=t#1s , Q=> , ET=> );

			tOff_RefreshRE(CLK:=tOff_Refresh.Q AND NOT bON,Q=>);
			IF tOff_RefreshRE.Q THEN
				byStep:= 20;
			END_IF

			IF bEnable THEN
				CASE byStep OF
				0:;
			
				10:
				sSendString:=CONCAT('LON','$R'); (*ON*)
				byStep:=0;

				20:
				sSendString:=CONCAT('LOFF','$R'); (*OFF*)
				byStep:=0;
			
			END_CASE

			END_IF

		(*Send String*)
		tOn_1s(IN:=NOT  tOn_1s.Q, PT:=t#1s , Q=> , ET=> );
		bSendString:=tOn_1s.Q;

		IF bSendString AND NOT fbSendString255.Busy THEN
		fbSendString255(
			SendString:=sSendString ,
			TXbuffer:=BufferWriteCom,
			Busy=>Busy ,
			Error=> Error);
		END_IF

		IF bON AND b1stBasketMemoryFlag THEN
		(*this will find where is the $R located in the string*)
		iReceivedStingProcess:=FIND(sReceivedStringRaw, sDelimiteChar);

		(*after you know the location, you can move the string to another string according to the size*)
		sReceivedString:=LEFT(sReceivedStringRaw, iReceivedStingProcess-1);

		ELSE

		sReceivedString := '';
		sReceivedStringRaw:='';

		END_IF


(*** for HandheldType Scanner***)
ELSIF  bHandHeldBarcodeScannerEn AND NOT bFixedTypeBarcodeScannerEn THEN

		tReceivedString_DelayReset(IN:= (sReceivedString <> '') AND NOT b1stBasketMemoryFlag , PT:=t#3.0s , Q=> , ET=> );

		IF bON_ForHandHeldTypeOnly (*AND b1stBasketMemoryFlag*) AND NOT tReceivedString_DelayReset.Q THEN
		(*this will find where is the $R located in the string*)
		iReceivedStingProcess:=FIND(sReceivedStringRaw, sDelimiteChar);

		(*after you know the location, you can move the string to another string according to the size*)
		sReceivedString:=LEFT(sReceivedStringRaw, iReceivedStingProcess-1);

		ELSIF tReceivedString_DelayReset.Q THEN

		sReceivedString:='';
		sReceivedStringRaw:='';

		ELSE

		sReceivedString:='';
		sReceivedStringRaw:='';

		END_IF

ELSE
		sReceivedString:='';
		sReceivedStringRaw:='';


END_IF

fbReceiveString(
	Prefix:='' ,
	Suffix:='$R',
	Timeout:=t#1s ,
	Reset:=fbReceiveString_Rst ,
	ReceivedString:=sReceivedStringRaw ,
	RXbuffer:=BufferReadCom ,
	StringReceived=>fbReceiveString_StrRcv ,
	Busy=> ,
	Error=> ,
	RxTimeout=> );

SerialLineControl(
	Mode:= SERIALLINEMODE_EL6_22B ,
	pComIn:= ADR(SerInDataCom) ,
	pComOut:= ADR(SerOutDataCom) ,
	SizeComIn:= SIZEOF(SerInDataCom),
	TxBuffer:= BufferWriteCom ,
	RxBuffer:= BufferReadCom,
	Error=> , 
	ErrorID=> );

END_FUNCTION_BLOCK

// ---- FBs/fbV3BarcodeCtrl/Sub FB/fb_V3StringEliminator.TcPOU
FUNCTION_BLOCK fb_V3StringEliminator
VAR_INPUT
	bEn: BOOL;
	sString: STRING;
	iCharEliminateQty : INT;
	iCharNeededQty: INT;
END_VAR
VAR_OUTPUT
	sResult: STRING;
	bDone : BOOL;
	bError: BOOL;
	sStatus: STRING(50);
END_VAR
VAR
	sResultTemp: STRING(50);
	iResultQty: INT;
	iLEN: INT;
	iPOS: INT;

END_VAR

iCharEliminateQty;


iLEN := LEN (sString);
iPOS := iCharEliminateQty+1;

IF bEn THEN
	sResultTemp := '';
	sResult := '';
	sStatus := '';
	bError := FALSE;
	bDone := FALSE;

	(*IF iCharNeededQty <= 0 THEN*)
	IF iLEN <= 0 THEN
		sResult := '';
		sStatus := 'Error - Character Needed Quantity Lower Than "0"';
		bError := TRUE;
		bDone := FALSE;


	ELSIF iCharEliminateQty >= 0 THEN
		sResultTemp := MID(sString, iLEN, iPOS);
		iResultQty := LEN(sResultTemp);
		sResult := sResultTemp;
		bDone := TRUE;
		sStatus := 'Done';

		IF  iLEN <  iPOS THEN
		sResult := '' ;
		sStatus := 'Error - Character Output Quantity Not Matched';
		bError := TRUE;
		bDone := FALSE;
		END_IF

	ELSE
	sResult := '';
	sStatus := 'Error - Character Eliminate Quantity Lower Than "0"';
	bError := TRUE;
	bDone := FALSE;
	END_IF

ELSE
	sResultTemp := '';
	sResult := '';
	sStatus := 'Press "bStart" to Execute';
	bError := FALSE;
	bDone := FALSE;
END_IF

END_FUNCTION_BLOCK

// ---- FBs/fbV3BarcodeCtrl/Sub FB/fb_V1BarcodeRegistration_UTAC.TcPOU
FUNCTION_BLOCK fb_V1BarcodeRegistration_UTAC
VAR_INPUT
END_VAR
VAR_OUTPUT
	sStatus : STRING;
END_VAR

VAR_IN_OUT
	sBarcodeInputFromScanner : STRING;
END_VAR
VAR
	iScanFL : INT;
	iFL : INT;
	iSFL : INT;
	ARbButtonRE : ARRAY [0..iBarcodeRegSecDisplayQty] OF R_TRIG;
	ARbBarcodeRegistrationEnRE : ARRAY [0..iBarcodeRegSecDisplayQty] OF R_TRIG;
	bBarcodeRegistrationEn : BOOL;
	bBarcodeDuplicate : BOOL;
	iRegNo: INT;
END_VAR

(*bBarcodeRegistrationEn button control - only one button ON at one time *)
iFL := 1;
	FOR iFL := 1 TO iBarcodeRegSecDisplayQty DO
		IF iFL >= 1 AND iFL <= iBarcodeRegSecDisplayQty THEN

			ARbButtonRE[iFL](CLK:=DsAr1sG_BarcodeRegSectionDisplayHMI[iFL].bBarcodeRegistrationEn , Q=> );

			IF ARbButtonRE[iFL].Q THEN
				iSFL := 1;
					FOR iSFL := 1 TO iBarcodeRegSecDisplayQty DO
						IF iSFL >= 1 AND iSFL <= iBarcodeRegSecDisplayQty THEN
							DsAr1sG_BarcodeRegSectionDisplayHMI[iSFL].bBarcodeRegistrationEn := FALSE;
						END_IF
					END_FOR
				DsAr1sG_BarcodeRegSectionDisplayHMI[iFL].bBarcodeRegistrationEn := TRUE;
			END_IF
		END_IF
	END_FOR


(*Reset sBarcodeRegistered when bBarcodeRegistrationEn enable*)
iScanFL := 1;
FOR iScanFL := 1 TO iBarcodeRegSecDisplayQty DO
	IF iScanFL >= 1 AND iScanFL <= iBarcodeRegSecDisplayQty THEN
		ARbBarcodeRegistrationEnRE[iScanFL](CLK:=DsAr1sG_BarcodeRegSectionDisplayHMI[iScanFL].bBarcodeRegistrationEn , Q=> );
		IF ARbBarcodeRegistrationEnRE[iScanFL].Q THEN
			DsAr1sG_BarcodeRegSectionDisplayHMI[iScanFL].sBarcodeRegistered := '';
			iRegNo := iScanFL;
			bBarcodeRegistrationEn := TRUE;
		END_IF

	END_IF
END_FOR


(*Reset bBarcodeRegistrationEn when iLinkProductRecipeNo and sBarcodeRegistered achieved*)
iScanFL := 1;
FOR iScanFL := 1 TO iBarcodeRegSecDisplayQty DO
	IF iScanFL >= 1 AND iScanFL <= iBarcodeRegSecDisplayQty THEN

		IF DsAr1sG_BarcodeRegSectionDisplayHMI[iScanFL].iLinkProductRecipeNo <> 0 AND DsAr1sG_BarcodeRegSectionDisplayHMI[iScanFL].sBarcodeRegistered <> '' AND DsAr1sG_BarcodeRegSectionDisplayHMI[iScanFL].bBarcodeRegistrationEn AND DsAr1sG_BarcodeRegSectionDisplayHMI[iScanFL].sLinkProductRecipeDescription <> '' THEN
			DsAr1sG_BarcodeRegSectionDisplayHMI[iScanFL].bBarcodeRegistrationEn := FALSE;
			bBarcodeRegistrationEn := FALSE;
			iRegNo := 0;
		END_IF

	END_IF
END_FOR

(*bBarcodeDuplicate function*)
bBarcodeDuplicate := FALSE;
IF bBarcodeRegistrationEn THEN
		iScanFL := 1;
		FOR iScanFL := 1 TO iBarcodeRegSecDisplayQty DO
			IF iScanFL >= 1 AND iScanFL <= iBarcodeRegSecDisplayQty THEN
				IF sBarcodeInputFromScanner <> '' THEN
					IF DsAr1sG_BarcodeRegSectionDisplayHMI[iScanFL].sBarcodeRegistered = sBarcodeInputFromScanner THEN
						bBarcodeDuplicate := TRUE;
					END_IF
				END_IF
			END_IF
		END_FOR
END_IF


(*Error Status shown when Barcode detected was ERROR*)
iScanFL := 1;
FOR iScanFL := 1 TO iBarcodeRegSecDisplayQty DO
	IF iScanFL >= 1 AND iScanFL <= iBarcodeRegSecDisplayQty THEN

		IF bBarcodeDuplicate AND DsAr1sG_BarcodeRegSectionDisplayHMI[iScanFL].bBarcodeRegistrationEn THEN
		sStatus := 'Error - Barcode Duplicated Found. Make sure assign barcode correctly';
		iScanFL := iBarcodeRegSecDisplayQty+1;
		ELSE
		sStatus := 'No Error Found';
		END_IF

	END_IF
END_FOR


(*
IF bBarcodeDuplicate AND bBarcodeRegistrationEn THEN
sStatus := 'Error - Barcode Duplicated Found. Make sure assign barcode correctly';
ELSE
sStatus := 'No Error Found';
END_IF
*)





(*Move sBarcodeInputFromScanner data into sBarcodeRegistered*)
iScanFL := 1;
FOR iScanFL := 1 TO iBarcodeRegSecDisplayQty DO
	IF iScanFL >= 1 AND iScanFL <= iBarcodeRegSecDisplayQty AND NOT bBarcodeDuplicate AND bBarcodeRegistrationEn THEN

		IF DsAr1sG_BarcodeRegSectionDisplayHMI[iScanFL].bBarcodeRegistrationEn AND sBarcodeInputFromScanner <> '' THEN
			DsAr1sG_BarcodeRegSectionDisplayHMI[iScanFL].sBarcodeRegistered := sBarcodeInputFromScanner;
		END_IF

	END_IF
END_FOR


(*Trace Product Recipe Description*)
IF iRegNo > 0 AND bBarcodeRegistrationEn AND DsAr1sG_BarcodeRegSectionDisplayHMI[iRegNo].iLinkProductRecipeNo > 0 THEN
	DsAr1sG_BarcodeRegSectionDisplayHMI[iRegNo].sLinkProductRecipeDescription := arProgramDescrip1[DsAr1sG_BarcodeRegSectionDisplayHMI[iRegNo].iLinkProductRecipeNo];
ELSIF  iRegNo > 0 AND bBarcodeRegistrationEn AND DsAr1sG_BarcodeRegSectionDisplayHMI[iRegNo].iLinkProductRecipeNo = 0 THEN
	DsAr1sG_BarcodeRegSectionDisplayHMI[iRegNo].sLinkProductRecipeDescription := '';
END_IF

END_FUNCTION_BLOCK

// ---- FBs/fbV3BarcodeCtrl/Sub FB/fb_V2BarcodeRegistration.TcPOU
FUNCTION_BLOCK fb_V2BarcodeRegistration
VAR_INPUT
END_VAR
VAR_OUTPUT
	sStatus : STRING;
END_VAR

VAR_IN_OUT
	sBarcodeInputFromScanner : STRING;
END_VAR
VAR
	iScanFL : INT;
	iFL : INT;
	iSFL : INT;
	ARbButtonRE : ARRAY [0..iBarcodeRegSecDisplayQty] OF R_TRIG;
	ARbBarcodeRegistrationEnRE : ARRAY [0..iBarcodeRegSecDisplayQty] OF R_TRIG;
	bBarcodeRegistrationEn : BOOL;
	bBarcodeDuplicate : BOOL;
	iRegNo: INT;
END_VAR

(*bBarcodeRegistrationEn button control - only one button ON at one time *)
iFL := 1;
	FOR iFL := 1 TO iBarcodeRegSecDisplayQty DO
		IF iFL >= 1 AND iFL <= iBarcodeRegSecDisplayQty THEN

			ARbButtonRE[iFL](CLK:=DsAr1sG_BarcodeRegSectionDisplayHMI[iFL].bBarcodeRegistrationEn , Q=> );

			IF ARbButtonRE[iFL].Q THEN
				iSFL := 1;
					FOR iSFL := 1 TO iBarcodeRegSecDisplayQty DO
						IF iSFL >= 1 AND iSFL <= iBarcodeRegSecDisplayQty THEN
							DsAr1sG_BarcodeRegSectionDisplayHMI[iSFL].bBarcodeRegistrationEn := FALSE;
						END_IF
					END_FOR
				DsAr1sG_BarcodeRegSectionDisplayHMI[iFL].bBarcodeRegistrationEn := TRUE;
			END_IF
		END_IF
	END_FOR


(*Reset sBarcodeRegistered when bBarcodeRegistrationEn enable*)
iScanFL := 1;
FOR iScanFL := 1 TO iBarcodeRegSecDisplayQty DO
	IF iScanFL >= 1 AND iScanFL <= iBarcodeRegSecDisplayQty THEN
		ARbBarcodeRegistrationEnRE[iScanFL](CLK:=DsAr1sG_BarcodeRegSectionDisplayHMI[iScanFL].bBarcodeRegistrationEn , Q=> );
		IF ARbBarcodeRegistrationEnRE[iScanFL].Q THEN
			DsAr1sG_BarcodeRegSectionDisplayHMI[iScanFL].sBarcodeRegistered := '';
			iRegNo := iScanFL;
			bBarcodeRegistrationEn := TRUE;
		END_IF

	END_IF
END_FOR


(*Reset bBarcodeRegistrationEn when iLinkProductRecipeNo and sBarcodeRegistered achieved*)
iScanFL := 1;
FOR iScanFL := 1 TO iBarcodeRegSecDisplayQty DO
	IF iScanFL >= 1 AND iScanFL <= iBarcodeRegSecDisplayQty THEN

		IF DsAr1sG_BarcodeRegSectionDisplayHMI[iScanFL].iLinkProductRecipeNo <> 0 AND DsAr1sG_BarcodeRegSectionDisplayHMI[iScanFL].sBarcodeRegistered <> '' AND DsAr1sG_BarcodeRegSectionDisplayHMI[iScanFL].bBarcodeRegistrationEn THEN
			DsAr1sG_BarcodeRegSectionDisplayHMI[iScanFL].bBarcodeRegistrationEn := FALSE;
			bBarcodeRegistrationEn := FALSE;
			iRegNo := 0;
		END_IF

	END_IF
END_FOR

(*bBarcodeDuplicate function*)
bBarcodeDuplicate := FALSE;
IF bBarcodeRegistrationEn THEN
		iScanFL := 1;
		FOR iScanFL := 1 TO iBarcodeRegSecDisplayQty DO
			IF iScanFL >= 1 AND iScanFL <= iBarcodeRegSecDisplayQty THEN
				IF sBarcodeInputFromScanner <> '' THEN
					IF DsAr1sG_BarcodeRegSectionDisplayHMI[iScanFL].sBarcodeRegistered = sBarcodeInputFromScanner THEN
						bBarcodeDuplicate := TRUE;
					END_IF
				END_IF
			END_IF
		END_FOR
END_IF


(*Error Status shown when Barcode detected was ERROR*)
iScanFL := 1;
FOR iScanFL := 1 TO iBarcodeRegSecDisplayQty DO
	IF iScanFL >= 1 AND iScanFL <= iBarcodeRegSecDisplayQty THEN

		IF bBarcodeDuplicate AND DsAr1sG_BarcodeRegSectionDisplayHMI[iScanFL].bBarcodeRegistrationEn THEN
		sStatus := 'Error - Barcode Duplicated Found. Make sure assign barcode correctly';
		iScanFL := iBarcodeRegSecDisplayQty+1;
		ELSE
		sStatus := 'No Error Found';
		END_IF

	END_IF
END_FOR


(*
IF bBarcodeDuplicate AND bBarcodeRegistrationEn THEN
sStatus := 'Error - Barcode Duplicated Found. Make sure assign barcode correctly';
ELSE
sStatus := 'No Error Found';
END_IF
*)





(*Move sBarcodeInputFromScanner data into sBarcodeRegistered*)
iScanFL := 1;
FOR iScanFL := 1 TO iBarcodeRegSecDisplayQty DO
	IF iScanFL >= 1 AND iScanFL <= iBarcodeRegSecDisplayQty AND NOT bBarcodeDuplicate AND bBarcodeRegistrationEn THEN

		IF DsAr1sG_BarcodeRegSectionDisplayHMI[iScanFL].bBarcodeRegistrationEn AND sBarcodeInputFromScanner <> '' THEN
			DsAr1sG_BarcodeRegSectionDisplayHMI[iScanFL].sBarcodeRegistered := sBarcodeInputFromScanner;
		END_IF

	END_IF
END_FOR


(*Trace Product Recipe Description*)
IF iRegNo > 0 AND bBarcodeRegistrationEn AND DsAr1sG_BarcodeRegSectionDisplayHMI[iRegNo].iLinkProductRecipeNo > 0 THEN
	DsAr1sG_BarcodeRegSectionDisplayHMI[iRegNo].sLinkProductRecipeDescription := arProgramDescrip1[DsAr1sG_BarcodeRegSectionDisplayHMI[iRegNo].iLinkProductRecipeNo];
ELSIF  iRegNo > 0 AND bBarcodeRegistrationEn AND DsAr1sG_BarcodeRegSectionDisplayHMI[iRegNo].iLinkProductRecipeNo = 0 THEN
	DsAr1sG_BarcodeRegSectionDisplayHMI[iRegNo].sLinkProductRecipeDescription := '';
END_IF

END_FUNCTION_BLOCK

// ---- FBs/fbV3BarcodeCtrl/Sub FB/fb_V3BarcodeTracer.TcPOU
FUNCTION_BLOCK fb_V3BarcodeTracer
VAR_INPUT
	bEn : BOOL;
(*	bfbV3En : BOOL;*)
	sTargetBarcode : STRING;
(*	ARsBarCodeRaw_V2 : ARRAY [0..99] OF STRING;
	ARsBarcodeDescrip_V2 : ARRAY [0..99] OF STRING;
*)

END_VAR
VAR_OUTPUT
	bBarcodeTraceSuccess : BOOL;
	bBarcodeTraceFail : BOOL;
	iBarcodeRecipeNo : INT;
	sBarcodeDescrip : STRING;

END_VAR
VAR
	i: INT;
	(*TracerRE : R_TRIG;*)

END_VAR

(*TracerRE(CLK:=bTracerST,Q=>);*)
IF NOT bEn THEN
	bBarcodeTraceSuccess := FALSE;
	bBarcodeTraceFail := FALSE;
	iBarcodeRecipeNo := 0;
	sBarcodeDescrip := '';
	i := 1;
END_IF

(* For V2 used*)
(*
IF NOT bfbV3En THEN

			IF bTracerST AND sTargetBarcode <> '' THEN
			bBarcodeTraceSuccess := FALSE;

					FOR i := 1 TO iProductRecipeArrayQty DO

					IF sTargetBarcode = ARsBarCodeRaw_V2[i] THEN
					sBarcodeInDescrip := ARsBarcodeDescrip_V2[i];
					iBarcodeInRecipeNo := i;
					bBarcodeTraceSuccess := TRUE;
					i := iProductRecipeArrayQty+1;
					END_IF
			
					END_FOR
			
			END_IF
			IF (i > iProductRecipeArrayQty AND bTracerST AND NOT bBarcodeTraceSuccess )THEN
			bBarcodeTraceFail := TRUE;
			ELSE
			bBarcodeTraceFail := FALSE;
			END_IF
END_IF
*)

(* For V3 used*)

IF TRUE(*bfbV3En*) THEN

			IF bEn AND sTargetBarcode <> '' THEN
			bBarcodeTraceSuccess := FALSE;

					FOR i := 1 TO iBarcodeRegQty DO

					IF sTargetBarcode = DsAr1sG_BarcodeRegistration[i].sBarcodeRegistered THEN
					sBarcodeDescrip := DsAr1sG_BarcodeRegistration[i].sLinkProductRecipeDescription ;
					iBarcodeRecipeNo := DsAr1sG_BarcodeRegistration[i].iLinkProductRecipeNo;
					bBarcodeTraceSuccess := TRUE;
					i := iBarcodeRegQty+1;
					END_IF

					END_FOR

			END_IF
			IF (i > iProductRecipeArrayQty AND bEn AND NOT bBarcodeTraceSuccess )THEN
			bBarcodeTraceFail := TRUE;
			ELSE
			bBarcodeTraceFail := FALSE;
			END_IF
END_IF

IF bBarcodeTraceFail THEN
iBarcodeRecipeNo := 0;
sBarcodeDescrip := '';
END_IF

END_FUNCTION_BLOCK

// ---- FBs/fbV3BarcodeCtrl/Sub FB/fb_V3BarcodeRegSectionDisplayController.TcPOU
FUNCTION_BLOCK fb_V3BarcodeRegSectionDisplayController

VAR_INPUT
	bEn : BOOL;
	bScrollUpPB : BOOL;
	bScrollDownPB : BOOL;
END_VAR

VAR_OUTPUT
	bUpEndFlag : BOOL;
	bDownEndFlag : BOOL;

END_VAR

VAR
	tSpeedUpTimer: TON;
	iScrollTimer: INT;
	tScrollTimer: TON;
	bScrollUpPBRE: R_TRIG;
	bScrollDownPBRE: R_TRIG;
	iFL: INT;
	bReadSection: BOOL;
	bTest: BOOL;

	iStep: INT;
	bENRE: R_TRIG;
END_VAR

VAR PERSISTENT
	iSectionDisplayInc : INT;
	iSectionDisplayIncBuffer: INT;

END_VAR

bENRE(CLK:=bEN , Q=> );

IF bEN THEN
iStep := 1;
ELSE
iStep := 0;
END_IF



CASE iStep OF

0:
bUpEndFlag:= FALSE;
bDownEndFlag:= FALSE;


1:
tSpeedUpTimer(IN:=(bScrollUpPB OR bScrollDownPB) AND NOT bScrollDownPBRE.Q AND NOT bScrollUpPBRE.Q , PT:=t#1.5s , Q=> , ET=> );
tScrollTimer(IN:=(bScrollUpPB OR bScrollDownPB) AND NOT tScrollTimer.Q , PT:=INT_TO_TIME(iScrollTimer) , Q=> , ET=> );

bScrollUpPBRE(CLK:=bScrollUpPB , Q=> );
bScrollDownPBRE(CLK:=bScrollDownPB , Q=> );

(*Scroll Speed Control*)
	IF NOT tSpeedUpTimer.Q THEN
		iScrollTimer := 500;
	ELSE
		IF iScrollTimer > 50 THEN
		iScrollTimer := iScrollTimer-1;
		END_IF
	END_IF

(*Scroll Up*)
	IF iSectionDisplayInc >= 1 THEN
		IF bScrollUpPBRE.Q OR (bScrollUpPB AND tScrollTimer.Q) THEN
			iSectionDisplayInc := iSectionDisplayInc -1;
		END_IF
	END_IF

(*Scroll Down*)
	IF iSectionDisplayInc <= (iBarcodeRegQty - iBarcodeRegSecDisplayQty - 1) THEN
		IF bScrollDownPBRE.Q OR (bScrollDownPB AND tScrollTimer.Q) THEN
			iSectionDisplayInc := iSectionDisplayInc +1;
		END_IF
	END_IF


(*Detect Inc Changed*)
	IF (iSectionDisplayInc <> iSectionDisplayIncBuffer) OR bENRE.Q THEN
		bReadSection := TRUE;
		iSectionDisplayIncBuffer := iSectionDisplayInc;
	END_IF


(*Read Section Exec*)
	IF bReadSection THEN
		iFL := 1;
			FOR iFL := 1 TO iBarcodeRegSecDisplayQty DO
				IF iFL >= 1 AND iFL <= iBarcodeRegSecDisplayQty THEN
					DsAr1sG_BarcodeRegSectionDisplayHMI[iFL] := DsAr1sG_BarcodeRegistration[iFL+iSectionDisplayInc];
				END_IF
			END_FOR
		bReadSection := FALSE;
	END_IF

(*Write Section Exec*)
	IF NOT bReadSection THEN
		iFL := 1;
			FOR iFL := 1 TO iBarcodeRegSecDisplayQty DO
				IF iFL >= 1 AND iFL <= iBarcodeRegSecDisplayQty THEN
					DsAr1sG_BarcodeRegistration[iFL+iSectionDisplayInc] := DsAr1sG_BarcodeRegSectionDisplayHMI[iFL];
				END_IF
			END_FOR

	END_IF

(*Generate Current Registration Number *)
		iFL := 1;
			FOR iFL := 1 TO iBarcodeRegSecDisplayQty DO
				IF iFL >= 1 AND iFL <= iBarcodeRegSecDisplayQty THEN
					iAr1sG_BarcodeRegNoSectionDisplayHMI[iFL] := iFL+iSectionDisplayInc;
				END_IF
			END_FOR


(*Up/Down End Flag*)
	IF iSectionDisplayInc = 0 THEN
		bUpEndFlag:= TRUE;
	ELSIF iSectionDisplayInc >= iBarcodeRegQty - iBarcodeRegSecDisplayQty THEN
		bDownEndFlag:= TRUE;
	ELSE
		bUpEndFlag:= FALSE;
		bDownEndFlag:= FALSE;
	END_IF

END_CASE


IF bTest THEN
iFL := 1;
	FOR iFL := 1 TO iBarcodeRegQty DO
		IF iFL >= 1 AND iFL <= iBarcodeRegQty THEN
			DsAr1sG_BarcodeRegistration[iFL].sBarcodeRegistered := CONCAT('Barcode', INT_TO_STRING(iFL));
		END_IF
	END_FOR
END_IF

END_FUNCTION_BLOCK

// ---- POUs/MainProgram/AutoProcessCtrl/BarcodeScanner.TcPOU
PROGRAM BarcodeScanner
VAR
	sBufferBarcodeScannerReceivedCmd: STRING;
	sStoreBarcodeScannerReceivedCmd: STRING;

	tLdConfirmDelayOnTimer: TON;
	bNewBarcodeDetected: BOOL;
	tNewBarcodeDetectedDelay: TON;

	iPushDescriptionFL: INT;
	sStringNIL: STRING;

	bBarcodeRegisterPBRE: R_TRIG;
	bBarcodeClearPBRE: R_TRIG;

	tLdSensor1DelayOffTimer: TON;
	tConveyorStartInternal: TON;

	bBarcodeValidFlag: BOOL;

	iFL: INT;

	tBarcodeData1 : TON;
	tBarcodeData2 : TON;
	tBarcodeData3 : TON;
	BarcodeData1RE: R_TRIG;
	BarcodeData2RE: R_TRIG;
	BarcodeData3RE: R_TRIG;

	bLdConveyorRapidRE: R_TRIG;
	bLdConveyorRapidHR: BOOL;
	bLdConveyorMotorFE: F_TRIG;
	
END_VAR

 (*****off for utac_barcode function*****)
(*COM(
	Mode:= SERIALLINEMODE_EL6_22B,
	pComIn:= ADR(SerInDataCom) ,
	pComOut:= ADR(SerOutDataCom),
	SizeComIn:= SIZEOF(SerInDataCom) ,
	TxBuffer:= BufferWriteCom,
	RxBuffer:= BufferReadCom,
	Error=> SerialComErrorFlag,
	ErrorID=> SerialComErrorID );
*)

COM1 (
	Mode:= SERIALLINEMODE_EL6_22B ,
	pComIn:= ADR(U485InData) ,
	pComOut:= ADR(U485OutData),
	SizeComIn:= SIZEOF(U485InData),
	TxBuffer:=U485BufferWrite ,
	RxBuffer:= U485BufferRead,
	Error=> SerialComErrorFlag1,
	ErrorID=> SerialComErrorID1 );
(*
ReceiveString(
	Prefix:= '',
	Suffix:= '$R',
	Timeout:=t#10s ,
	Reset:=fbReceiveString_Rst ,
	ReceivedString:=sBarcodeScannerReceived ,
	RXbuffer:= BufferReadCom,
	StringReceived=> fbReceiveString_StrRcv,
	Busy=> ,
	Error=> ,
	RxTimeout=> );
*)

presuffix(
	bEN:= TRUE,
	bPrefixEliminatorEN:= FALSE,
	bSuffixEliminatorEN:= TRUE,
	sData:= dsSerialCom.sReceivedString ,
	sPrefix:= '',
	sSuffix:= '$R',
	iLengthAfterPrefix:= 0,
	iLengthBeforeSuffix:=ilengthElimater,
	sPrefixEliminatorResult=> ,
	sSuffixEliminatorResult=>sBarcodeScannerReceivedResult,
	sPreSuffixEliminatorResult=> ,
	sNoneEliminatorReseult=> );


IF sBarcodeScannerReceivedCmd = Empty THEN
bBarcodeEmpty := TRUE;
ELSE
bBarcodeEmpty := FALSE;
END_IF
(*
(*(*****off for utac_barcode function*****)*)
BarcodeTracer(
	bTracerST:= tNewBarcodeDetectedDelay.Q,
	sTargetBarcode:= sBarcodeScannerReceivedCmd,
	AR99sBarCodeRaw:= ARsBarcodeOutput,
	AR99sBarcodeDescrip:= ARsProgramDescrip,
	bBarcodeTraceSuccess=>bBarcodeValid ,
	bBarcodeTraceFail=> bBarcodeInvalid,
	iBarcodeInRecipeNo=> BarcodeRecipeNO,
	sBarcodeInDescrip=> sBarcodeDescripOut);
*)

(*Check if Barcode scanner data change*)

tNewBarcodeDetectedDelay(IN:= sBarcodeScannerReceivedCmd = sBufferBarcodeScannerReceivedCmd AND sBarcodeScannerReceivedCmd <> '' ,PT:=t#1s, Q=> , ET=> );

IF sBarcodeScannerReceivedCmd <> sBufferBarcodeScannerReceivedCmd AND  sBarcodeScannerReceivedCmd <> ''THEN
sStoreBarcodeScannerReceivedCmd := sBarcodeScannerReceivedCmd;
sBufferBarcodeScannerReceivedCmd := sBarcodeScannerReceivedCmd;
bNewBarcodeDetected := TRUE;
END_IF

ClearBufferTime(IN:= ManualTest OR bBarcodeBypass, PT:= t#0.1s , Q=> , ET=> );
IF ClearBufferTime.Q THEN
sBarcodeScannerReceived := '';
sBasketNo:='';
END_IF

(* Loading Basket Confirm Bit Delay On Control *)

IF iBarcodeRecipeNo_OUT <> 0 AND sBarcodeDescrip_OUT <> '' (*ARsHMIBarcodeData_ScanIn[1]  <> '' AND ARsHMIBarcodeData_ScanIn[2]  <> '' AND ARsHMIBarcodeData_ScanIn[3]  <> ''*) THEN
bBarcodeValidFlag := TRUE;
END_IF

IF bBarcodeValidFlag AND bBarcodeValid AND bBarcodeConfirm THEN
bConfirmPB		   := TRUE;
END_IF

IF NOT ARbDI[eX14000_LoadingConveyorSensor_Feed] THEN
bBarcodeValidFlag := FALSE;
bConfirmPB		   := FALSE;
END_IF



(***** Loading Basket Memory*******)
tLdSensor1DelayOffTimer(IN:=(NOT ARbDI[eX14000_LoadingConveyorSensor_Feed] ) , PT:= T#3S, Q=> , ET=> );

IF tLdSensor1DelayOffTimer.Q THEN
sBarcodeScannerReceived := '' ;
AR2sDSCv_LdConfirmBasketInfo[1,1].iProductRecipeNo := 0;
sBasketNo := '';
ARbBarcodeStorageEnable[1] := FALSE;
ARbBarcodeStorageEnable[2] := FALSE;
ARbBarcodeStorageEnable[3] := FALSE;
sBasketNo:='';
END_IF

IF NOT ARbDI[eX14000_LoadingConveyorSensor_Feed] THEN
sBasketNo:='';
END_IF
(*
tBarcodeData1(IN:= ARsHMIBarcodeData_ScanIn[1] <> '', PT:= t#0.5s, Q=> , ET=> );
tBarcodeData2(IN:= ARsHMIBarcodeData_ScanIn[2] <> '', PT:= t#0.5s, Q=> , ET=> );
tBarcodeData3(IN:= ARsHMIBarcodeData_ScanIn[3] <> '', PT:= t#0.5s, Q=> , ET=> );

BarcodeData1RE(CLK:= tBarcodeData1.Q, Q=> );
BarcodeData2RE(CLK:= tBarcodeData2.Q, Q=> );
BarcodeData3RE(CLK:= tBarcodeData3.Q, Q=> );

IF BarcodeData1RE.Q THEN
ARbBarcodeStorageEnable[1] := FALSE;
END_IF

IF BarcodeData2RE.Q THEN
ARbBarcodeStorageEnable[2] := FALSE;
END_IF

IF BarcodeData3RE.Q THEN
ARbBarcodeStorageEnable[3] := FALSE;
END_IF
*)
IF tLdSensor1DelayOffTimer.Q AND (NOT ManualPageEnable OR NOT bAllowLoadingBasketIn) THEN
iUserDefineProductRecipeNo := 0;
iBarcodeRecipeNo_OUT := 0;
END_IF


tLdConfirmDelayOnTimer(IN:= (bMainOnOff(*bAutoStartPb*) OR ManualPageEnable) AND ((bConfirmPB OR  iSecs_Control_State=5  AND NOT bBarcodeBypass) OR ( bBarcodeBypass)) AND (ARbDI[eX14000_LoadingConveyorSensor_Feed]), PT:= T#3S, Q=> , ET=> );
(*Note-iSecs_Control_State<>5 is when SEcs\Gem Remote is Enable*)
IF tLdConfirmDelayOnTimer.Q THEN
	IF NOT bBarcodeBypass AND iSecs_Control_State<>5 THEN
	AR2sDSCv_LdConfirmBasketInfo[1,1].iProductRecipeNo 		:= (*BarcodeRecipeNO*)iBarcodeRecipeNo_OUT;
	AR2sDSCv_LdConfirmBasketInfo[1,1].ARsBarcodeData[1] 	:= sBarcodeScannerReceivedCmd;
	AR2sDSCv_LdConfirmBasketInfo[1,1].ARsBarcodeData[2] 	:= sBasketNo;
	AR2sDSCv_LdConfirmBasketInfo[1,1].ARsBarcodeData[3] 	:= ARsBarcodeData_LdBasketInfo[3];
	AR2sDSCv_LdConfirmBasketInfo[1,1].sProgramDescription 	:= (*sBarcodeDescripOut*)sBarcodeDescrip_OUT;

	ELSIF bBarcodeBypass AND iSecs_Control_State<>5 THEN
	AR2sDSCv_LdConfirmBasketInfo[1,1].iProductRecipeNo 		:= iUserDefineProductRecipeNo;
	AR2sDSCv_LdConfirmBasketInfo[1,1].ARsBarcodeData[1] 	:= INT_TO_STRING(iUserDefineProductRecipeNo);
	AR2sDSCv_LdConfirmBasketInfo[1,1].ARsBarcodeData[2] 	:= '0';
	AR2sDSCv_LdConfirmBasketInfo[1,1].ARsBarcodeData[3] 	:= '0';
	AR2sDSCv_LdConfirmBasketInfo[1,1].sProgramDescription 	:= ARsProductRecipeDescription[iUserDefineProductRecipeNo];

	ELSIF  iSecs_Control_State=5 THEN
	AR2sDSCv_LdConfirmBasketInfo[1,1].iProductRecipeNo 		:= iServerSecsGemProgNo;
	AR2sDSCv_LdConfirmBasketInfo[1,1].ARsBarcodeData[1] 	:= sBarcodeScannerReceivedCmd;
	AR2sDSCv_LdConfirmBasketInfo[1,1].ARsBarcodeData[2] 	:= ARsBarcodeData_LdBasketInfo[2];
	AR2sDSCv_LdConfirmBasketInfo[1,1].ARsBarcodeData[3] 	:= ARsBarcodeData_LdBasketInfo[3];
	AR2sDSCv_LdConfirmBasketInfo[1,1].sProgramDescription 	:= sBarcodeDescrip_OUT;
	END_IF

END_IF
(*
iFL := 1;
FOR iFL := 1 TO iCvLdQty DO
	IF iFL >= 1 AND iFL <= iCvLdQty THEN

		IF AR2sDSCv_LdConfirmBasketInfo[1,iFL].ARsBarcodeData[3] <> '' THEN
		ARbLdBasketBarcodeAvailable[iFL] := TRUE;
		ELSE
		ARbLdBasketBarcodeAvailable[iFL] := FALSE;
		END_IF
	END_IF
END_FOR





(* Clear Barcode Scanner Data Bit Control *)
Trig2(CLK:= bClearData, Q=> );

IF Trig2.Q THEN
sBarcodeScannerReceivedCmd := '' ;
END_IF
(*
IF NOT bBarcodeBypass THEN
BarcodeByPassNo := 0;
END_IF
*)
(* Ld Basket Confirm Memory and Barcode Data Control *)

bBarcodeSortingEn := X150_00;

fbBarcodeSorting10ML5575(
	bEN:= bBarcodeSortingEn,
	bBarcodeTracerInvalidFlag:= bBarcodeInvalid ,
	bConfirmPB:= bConfirmPB,
	ARbBarcodeStorageEnable:= ARbBarcodeStorageEnable,
	sBarcodeInputFromScanner:= sBarcodeScannerReceivedCmd ,
	ARbHMIBarcodeScanEn:= ARbHMIBarcodeScanEn,
	ARsHMIBarcodeData_ScanIn:= ARsHMIBarcodeData_ScanIn,
	ARsBarcodeData_LdBasketInfo:= ARsBarcodeData_LdBasketInfo,
	bBarcodeScanEnableFlag=> bBarcodeScanEnableFlag,
	bConfirmReadyFlag=> bConfirmReadyFlag );

(*Push the Product Recipe Description out to AR99 for Barcode register used*)

iPushDescriptionFL := 1;
	IF iPushDescriptionFL > 0 AND iPushDescriptionFL <= iProductRecipeArrayQty THEN
		FOR iPushDescriptionFL := 1 TO iProductRecipeArrayQty DO
		ARsProgramDescrip[iPushDescriptionFL] := PnPstorageMemory_Arm.fbGnrProductRecipeMemory_Main.fbA1PnpSequenceMemory.ARsStoragePnpSequenceDescription[iPushDescriptionFL];
		END_FOR
	END_IF

bBarcodeRegisterPBRE(CLK:=bBarcodeRegisterPB , Q=> );
IF bBarcodeRegisterPBRE.Q THEN
	IF iBarcodeRegisterProductNo > 0 AND iBarcodeRegisterProductNo <= iProductRecipeArrayQty THEN
	ARsBarcodeOutput[iBarcodeRegisterProductNo] := ARsHMIBarcodeData_ScanIn[3]; (*sStoreBarcodeScannerReceivedCmd;*)
	ARsBarcodeBatch[iBarcodeRegisterProductNo] := ARsHMIBarcodeData_ScanIn[1];
	ARsBarcodeJob[iBarcodeRegisterProductNo] := ARsHMIBarcodeData_ScanIn[2];
	END_IF
END_IF

bBarcodeClearPBRE(CLK:=bBarcodeClearPB , Q=> );
IF bBarcodeClearPBRE.Q THEN
	IF iBarcodeRegisterProductNo > 0 AND iBarcodeRegisterProductNo <= iProductRecipeArrayQty THEN
	ARsBarcodeOutput[iBarcodeRegisterProductNo] := '';
	ARsBarcodeBatch[iBarcodeRegisterProductNo] := '';
	ARsBarcodeJob[iBarcodeRegisterProductNo] := '';
	END_IF
END_IF
*)

END_PROGRAM

// ---- POUs/MainProgram/AutoSevenDayOnOffCtrl/SevenDayCtrl.TcPOU
PROGRAM SevenDayCtrl
VAR

	SevenDayOn: fbSevenDaySys;
	SevenDayOff: fbSevenDaySys;

END_VAR

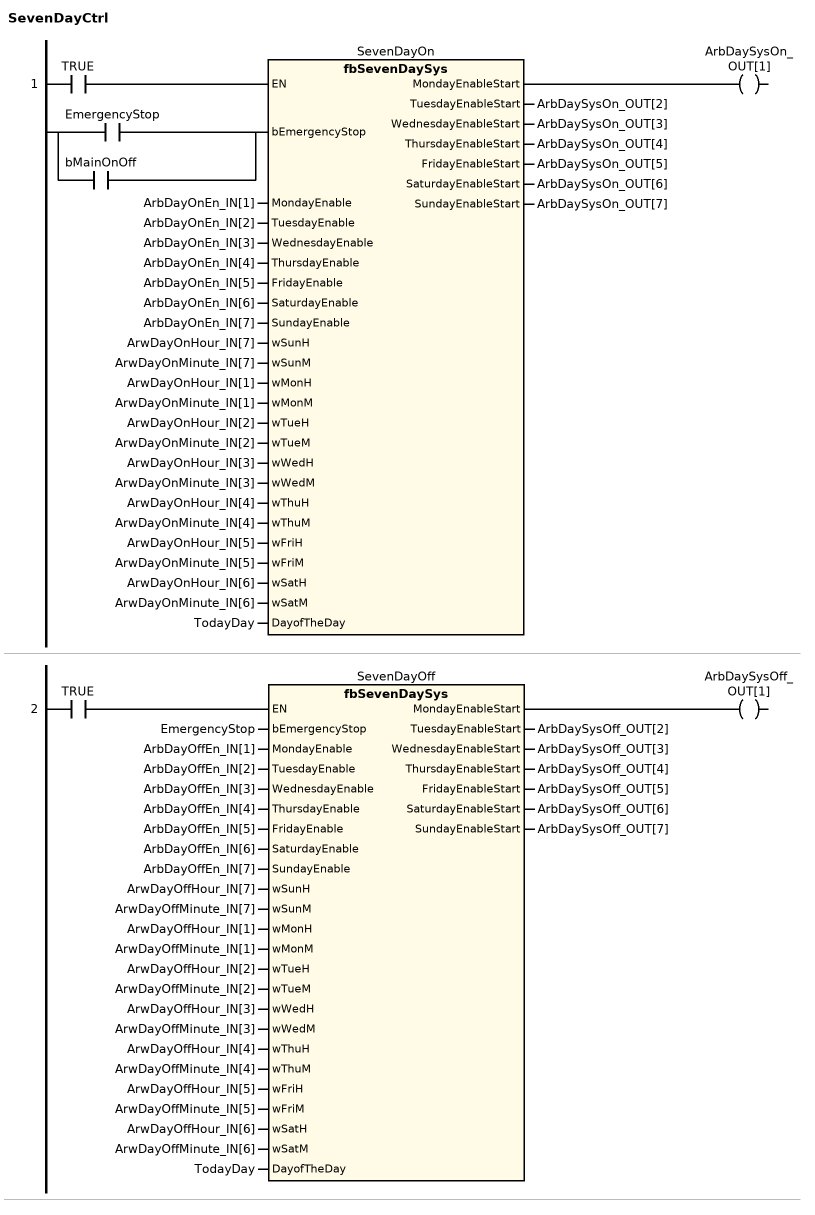
// NETWORK 1
SevenDayOn(
    bEmergencyStop := EmergencyStop OR bMainOnOff,
    MondayEnable := ArbDayOnEn_IN[1],
    TuesdayEnable := ArbDayOnEn_IN[2],
    WednesdayEnable := ArbDayOnEn_IN[3],
    ThursdayEnable := ArbDayOnEn_IN[4],
    FridayEnable := ArbDayOnEn_IN[5],
    SaturdayEnable := ArbDayOnEn_IN[6],
    SundayEnable := ArbDayOnEn_IN[7],
    wSunH := ArwDayOnHour_IN[7],
    wSunM := ArwDayOnMinute_IN[7],
    wMonH := ArwDayOnHour_IN[1],
    wMonM := ArwDayOnMinute_IN[1],
    wTueH := ArwDayOnHour_IN[2],
    wTueM := ArwDayOnMinute_IN[2],
    wWedH := ArwDayOnHour_IN[3],
    wWedM := ArwDayOnMinute_IN[3],
    wThuH := ArwDayOnHour_IN[4],
    wThuM := ArwDayOnMinute_IN[4],
    wFriH := ArwDayOnHour_IN[5],
    wFriM := ArwDayOnMinute_IN[5],
    wSatH := ArwDayOnHour_IN[6],
    wSatM := ArwDayOnMinute_IN[6],
    DayofTheDay := TodayDay,
    TuesdayEnableStart => ArbDaySysOn_OUT[2],
    WednesdayEnableStart => ArbDaySysOn_OUT[3],
    ThursdayEnableStart => ArbDaySysOn_OUT[4],
    FridayEnableStart => ArbDaySysOn_OUT[5],
    SaturdayEnableStart => ArbDaySysOn_OUT[6],
    SundayEnableStart => ArbDaySysOn_OUT[7]); // fbSevenDaySys
ArbDaySysOn_OUT[1] := SevenDayOn.MondayEnableStart;

// NETWORK 2
SevenDayOff(
    bEmergencyStop := EmergencyStop,
    MondayEnable := ArbDayOffEn_IN[1],
    TuesdayEnable := ArbDayOffEn_IN[2],
    WednesdayEnable := ArbDayOffEn_IN[3],
    ThursdayEnable := ArbDayOffEn_IN[4],
    FridayEnable := ArbDayOffEn_IN[5],
    SaturdayEnable := ArbDayOffEn_IN[6],
    SundayEnable := ArbDayOffEn_IN[7],
    wSunH := ArwDayOffHour_IN[7],
    wSunM := ArwDayOffMinute_IN[7],
    wMonH := ArwDayOffHour_IN[1],
    wMonM := ArwDayOffMinute_IN[1],
    wTueH := ArwDayOffHour_IN[2],
    wTueM := ArwDayOffMinute_IN[2],
    wWedH := ArwDayOffHour_IN[3],
    wWedM := ArwDayOffMinute_IN[3],
    wThuH := ArwDayOffHour_IN[4],
    wThuM := ArwDayOffMinute_IN[4],
    wFriH := ArwDayOffHour_IN[5],
    wFriM := ArwDayOffMinute_IN[5],
    wSatH := ArwDayOffHour_IN[6],
    wSatM := ArwDayOffMinute_IN[6],
    DayofTheDay := TodayDay,
    TuesdayEnableStart => ArbDaySysOff_OUT[2],
    WednesdayEnableStart => ArbDaySysOff_OUT[3],
    ThursdayEnableStart => ArbDaySysOff_OUT[4],
    FridayEnableStart => ArbDaySysOff_OUT[5],
    SaturdayEnableStart => ArbDaySysOff_OUT[6],
    SundayEnableStart => ArbDaySysOff_OUT[7]); // fbSevenDaySys
ArbDaySysOff_OUT[1] := SevenDayOff.MondayEnableStart;

END_PROGRAM

// ---- FBs/B_JKS_NewFB/FBP-SevenDayAutoOnOff/fbSevenDaySys.TcPOU
FUNCTION_BLOCK fbSevenDaySys
VAR_INPUT

	bEmergencyStop : BOOL;

	MondayEnable: BOOL;
	TuesdayEnable: BOOL;
	WednesdayEnable: BOOL;
	ThursdayEnable: BOOL;
	FridayEnable: BOOL;
	SaturdayEnable: BOOL;
	SundayEnable: BOOL;

	wSunH : WORD;
	wSunM : WORD;
	wMonH : WORD;
	wMonM : WORD;
	wTueH : WORD;
	wTueM : WORD;
	wWedH : WORD;
	wWedM : WORD;
	wThuH : WORD;
	wThuM : WORD;
	wFriH : WORD;
	wFriM : WORD;
	wSatH : WORD;
	wSatM: WORD;


END_VAR

VAR_IN_OUT

	DayofTheDay: STRING;

END_VAR

VAR_OUTPUT


	MondayEnableStart: BOOL;
	TuesdayEnableStart: BOOL;
	WednesdayEnableStart: BOOL;
	ThursdayEnableStart: BOOL;
	FridayEnableStart: BOOL;
	SaturdayEnableStart: BOOL;
	SundayEnableStart: BOOL;

END_VAR
VAR

	LocalSystemTime:FB_LocalSystemTime;
	SysTime:TIMESTRUCT;
	wHour: WORD;
	wMin: WORD;
	wSec: WORD;
	wDayOfWeek: WORD;
	wDate: WORD;

	bDailyRefresh: BOOL;
	SundayEnableStartInt: BOOL;
	SaturdayEnableStartint: BOOL;
	FridayEnableStartint: BOOL;
	ThursdayEnableStartint: BOOL;
	WednesdayEnableStartint: BOOL;
	TuesdayEnableStartint: BOOL;
	MondayEnableStartint: BOOL;
	MondayEnableStartRE: R_TRIG;
	TuesdayEnableStartRE: R_TRIG;
	WednesdayEnableStartRE: R_TRIG;
	ThursdayEnableStartRE: R_TRIG;
	FridayEnableStartRE: R_TRIG;
	SaturdayEnableStartRE: R_TRIG;
	SundayEnableStartRE: R_TRIG;
END_VAR

LocalSystemTime(
	sNetID:='' ,
	bEnable:=TRUE ,
	dwCycle:= ,
	dwOpt:= ,
	tTimeout:= ,
	bValid=> ,
	systemTime=>SysTime,
	tzID=> );

wDate:=SysTime.wDay;
wDayOfWeek:=SysTime.wDayOfWeek;
wHour:=SysTime.wHour;
wMin:=SysTime.wMinute;
wSec:=SysTime.wSecond;


(*Display today day*)
(*=========================================================================*)
IF wDayOfWeek =1 THEN
	DayofTheDay:='Monday';

END_IF

IF wDayOfWeek =2 THEN
	DayofTheDay:='Tuesday';
END_IF

IF wDayOfWeek =3 THEN
	DayofTheDay:='Wednesday';
END_IF

IF wDayOfWeek =4 THEN
	DayofTheDay:='Thursday';
END_IF

IF wDayOfWeek =5 THEN
	DayofTheDay:='Friday';
END_IF

IF wDayOfWeek =6 THEN
	DayofTheDay:='Saturday';
END_IF

IF wDayOfWeek =7 THEN
	DayofTheDay:='Sunday';
END_IF
(*=========================================================================*)
(*
IF wHour = 0 THEN
bDailyRefresh := TRUE;
END_IF

IF bEmergencyStop THEN
bDailyRefresh := FALSE;
END_IF
*)

(*Timer Count up*)
(*===========================================================================*)
MondayEnableStartRE(CLK:=MondayEnableStartint , Q=> );
TuesdayEnableStartRE(CLK:=TuesdayEnableStartint , Q=> );
WednesdayEnableStartRE(CLK:=WednesdayEnableStartint , Q=> );
ThursdayEnableStartRE(CLK:=ThursdayEnableStartint , Q=> );
FridayEnableStartRE(CLK:=FridayEnableStartint , Q=> );
SaturdayEnableStartRE(CLK:=SaturdayEnableStartint , Q=> );
SundayEnableStartRE(CLK:=SundayEnableStartint , Q=> );

IF MondayEnableStartRE.Q THEN
MondayEnableStart := TRUE;
END_IF
IF TuesdayEnableStartRE.Q THEN
TuesdayEnableStart := TRUE;
END_IF
IF WednesdayEnableStartRE.Q THEN
WednesdayEnableStart := TRUE;
END_IF
IF ThursdayEnableStartRE.Q THEN
ThursdayEnableStart := TRUE;
END_IF
IF FridayEnableStartRE.Q THEN
FridayEnableStart := TRUE;
END_IF
IF SaturdayEnableStartRE.Q THEN
SaturdayEnableStart := TRUE;
END_IF
IF SundayEnableStartRE.Q THEN
SundayEnableStart := TRUE;
END_IF

IF	MondayEnable
	AND DayofTheDay='Monday'
	AND wMonH =wHour
	AND wMonM = wMin THEN
	MondayEnableStartint:=TRUE;
END_IF

IF 	NOT MondayEnable
	OR bEmergencyStop THEN
	MondayEnableStartint:=FALSE;
	MondayEnableStart:=FALSE;
END_IF


IF	TuesdayEnable
	AND DayofTheDay='Tuesday'
	AND wTueH =wHour
	AND wTueM = wMin THEN
	TuesdayEnableStartint:=TRUE;
END_IF


IF 	NOT TuesdayEnable
	OR bEmergencyStop THEN
	TuesdayEnableStartint:=FALSE;
	TuesdayEnableStart:=FALSE;
END_IF


IF	WednesdayEnable
	AND DayofTheDay='Wednesday'
	AND wWedH =wHour
	AND wWedM = wMin THEN
	WednesdayEnableStartint:=TRUE;
END_IF


IF 	NOT WednesdayEnable
	OR bEmergencyStop  THEN
	WednesdayEnableStartint:=FALSE;
	WednesdayEnableStart:=FALSE;
END_IF


IF	ThursdayEnable
	AND DayofTheDay='Thursday'
	AND wThuH =wHour
	AND wThuM = wMin THEN
	ThursdayEnableStartint:=TRUE;
END_IF


IF 	NOT ThursdayEnable
	OR bEmergencyStop  THEN
	ThursdayEnableStartint:=FALSE;
	ThursdayEnableStart:=FALSE;
END_IF


IF	FridayEnable
	AND DayofTheDay='Friday'
	AND wFriH =wHour
	AND wFriM = wMin THEN
	FridayEnableStartint:=TRUE;
END_IF


IF 	NOT FridayEnable
	OR bEmergencyStop THEN
	FridayEnableStartint:=FALSE;
	FridayEnableStart:=FALSE;
END_IF


IF	SaturdayEnable
	AND DayofTheDay='Saturday'
	AND wSatH =wHour
	AND wSatM = wMin THEN
	SaturdayEnableStartint:=TRUE;
END_IF


IF 	NOT SaturdayEnable
	OR bEmergencyStop  THEN
	SaturdayEnableStartint:=FALSE;
	SaturdayEnableStart:=FALSE;
END_IF


IF	SundayEnable
	AND DayofTheDay='Sunday'
	AND wSunH =wHour
	AND wSunM = wMin THEN
	SundayEnableStartInt:=TRUE;
END_IF


IF 	NOT SundayEnable
	OR bEmergencyStop THEN
	SundayEnableStartint:=FALSE;
	SundayEnableStart:=FALSE;
END_IF

END_FUNCTION_BLOCK

// ---- POUs/MainProgram/AutoSevenDayOnOffCtrl/SevenDayOnOffConf.TcPOU
PROGRAM SevenDayOnOffConf
VAR

	bOver2ndLimitAlarmOccur: BOOL;


END_VAR

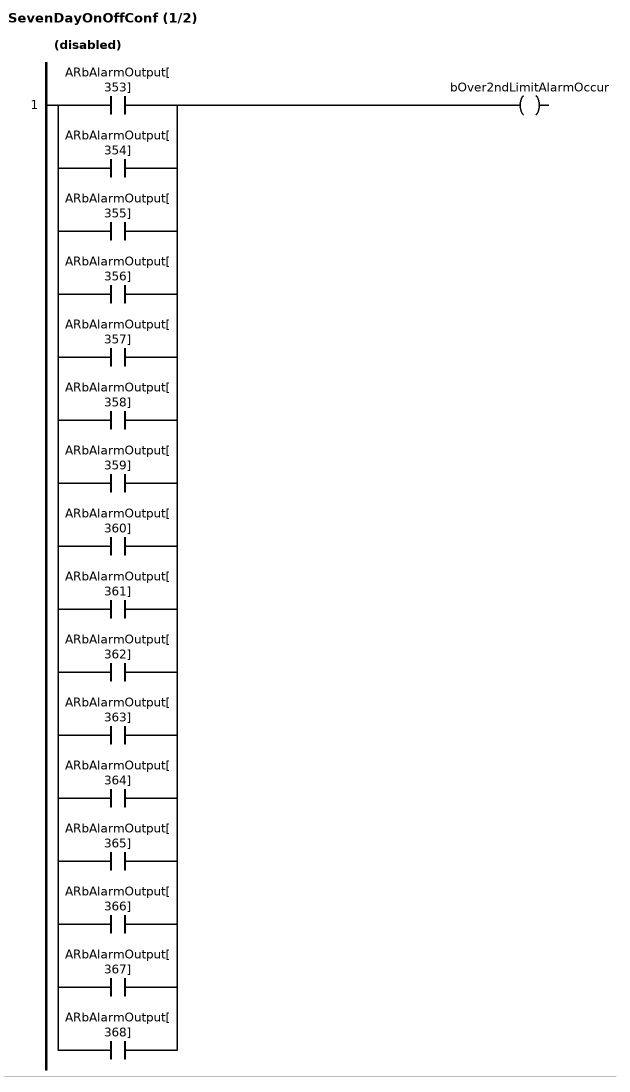
// NETWORK 1 (disabled)
// bOver2ndLimitAlarmOccur := ARbAlarmOutput[353] OR ARbAlarmOutput[354] OR ARbAlarmOutput[355] OR ARbAlarmOutput[356] OR ARbAlarmOutput[357] OR ARbAlarmOutput[358] OR ARbAlarmOutput[359] OR ARbAlarmOutput[360] OR ARbAlarmOutput[361] OR ARbAlarmOutput[362] OR ARbAlarmOutput[363] OR ARbAlarmOutput[364] OR ARbAlarmOutput[365] OR ARbAlarmOutput[366] OR ARbAlarmOutput[367] OR ARbAlarmOutput[368];

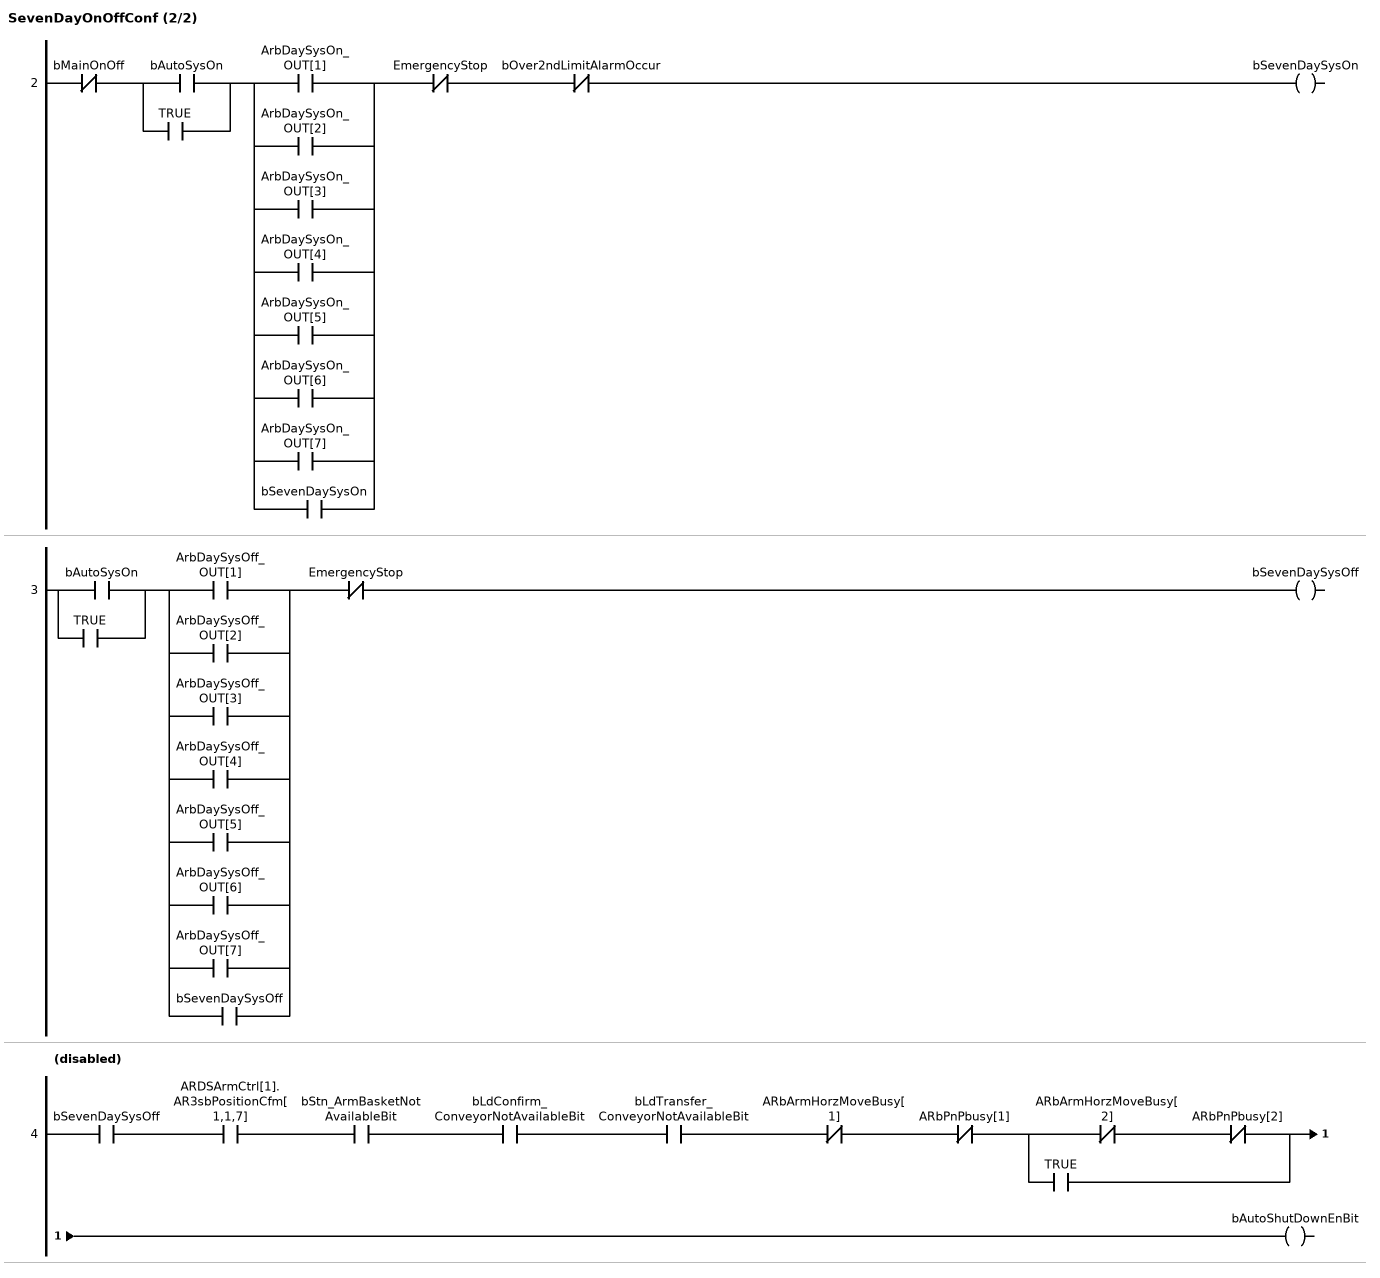
// NETWORK 2
bSevenDaySysOn := (NOT bMainOnOff AND (bAutoSysOn OR TRUE) AND (ArbDaySysOn_OUT[1] OR ArbDaySysOn_OUT[2] OR ArbDaySysOn_OUT[3] OR ArbDaySysOn_OUT[4] OR ArbDaySysOn_OUT[5] OR ArbDaySysOn_OUT[6] OR ArbDaySysOn_OUT[7] OR bSevenDaySysOn)) AND NOT EmergencyStop AND NOT bOver2ndLimitAlarmOccur;

// NETWORK 3
bSevenDaySysOff := ((bAutoSysOn OR TRUE) AND (ArbDaySysOff_OUT[1] OR ArbDaySysOff_OUT[2] OR ArbDaySysOff_OUT[3] OR ArbDaySysOff_OUT[4] OR ArbDaySysOff_OUT[5] OR ArbDaySysOff_OUT[6] OR ArbDaySysOff_OUT[7] OR bSevenDaySysOff)) AND NOT EmergencyStop;

// NETWORK 4 (disabled)
// bAutoShutDownEnBit := bSevenDaySysOff AND ARDSArmCtrl[1].AR3sbPositionCfm[1,1,7] AND bStn_ArmBasketNotAvailableBit AND bLdConfirm_ConveyorNotAvailableBit AND bLdTransfer_ConveyorNotAvailableBit AND NOT ARbArmHorzMoveBusy[1] AND NOT ARbPnPbusy[1] AND (NOT ARbArmHorzMoveBusy[2] AND NOT ARbPnPbusy[2] OR TRUE);

END_PROGRAM

// ---- POUs/MainProgram/BaseWork/TowerLightCtrl.TcPOU
PROGRAM TowerLightCtrl
VAR
	TLctrl					: fbTowerLightCtrl;
	CLKPLS					: CLOCK_PLS;
	CP						: BOOL;
	SFQ						: BOOL;

	ARbAlarmOutput421RE		: R_TRIG;
	ARbAlarmOutput422RE		: R_TRIG;
	ARbAlarmOutput424RE		: R_TRIG;
	ARbAlarmOutput425RE		: R_TRIG;
	ARbAlarmOutput113RE		: R_TRIG;

	ARbAlarmOutput423RE		: R_TRIG;
	ARbAlarmOutput426RE		: R_TRIG;
	ARbAlarmOutput429RE		: R_TRIG;

	bAlarmOccurFlagIND		: BOOL;
	bBuzzerFlagIND			: BOOL;

END_VAR
VAR // added by the converter: edge detectors and wires of the graphical bodies
    _w1 : BOOL;
END_VAR

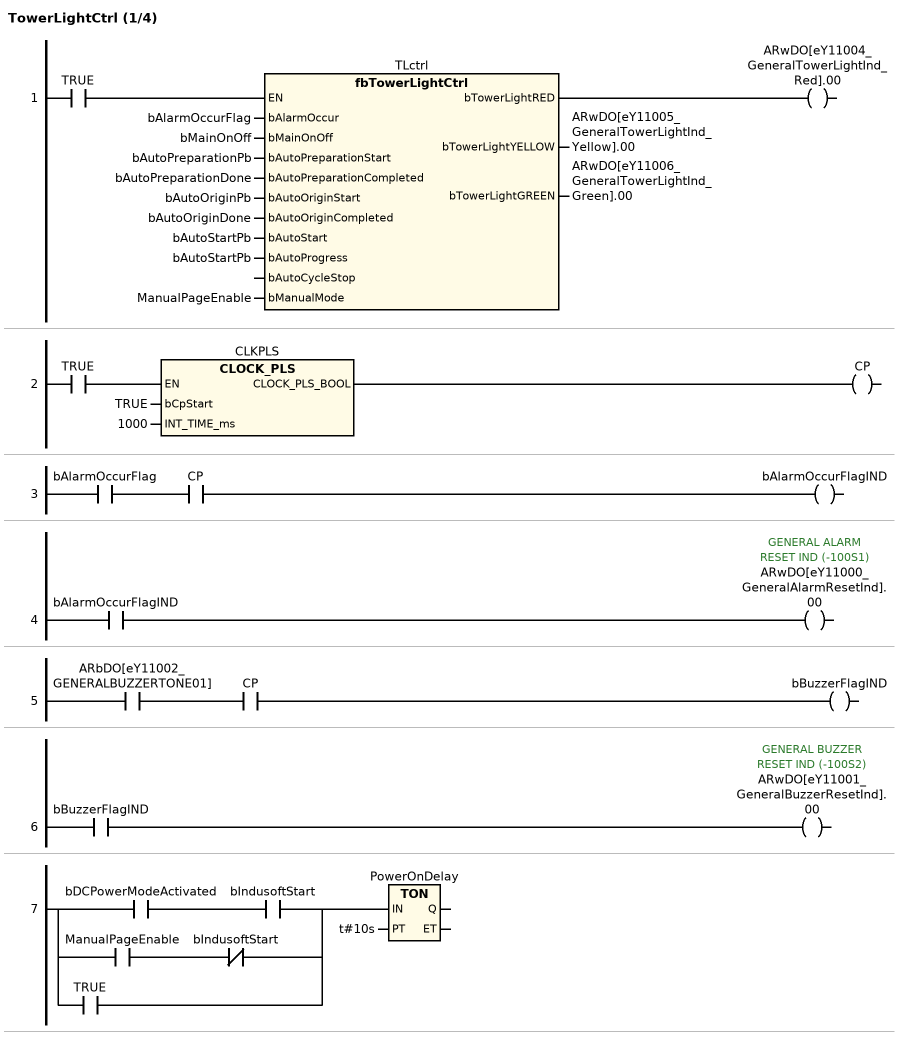
// NETWORK 1
TLctrl(
    bAlarmOccur := bAlarmOccurFlag,
    bMainOnOff := bMainOnOff,
    bAutoPreparationStart := bAutoPreparationPb,
    bAutoPreparationCompleted := bAutoPreparationDone,
    bAutoOriginStart := bAutoOriginPb,
    bAutoOriginCompleted := bAutoOriginDone,
    bAutoStart := bAutoStartPb,
    bAutoProgress := bAutoStartPb,
    bManualMode := ManualPageEnable,
    bTowerLightYELLOW => ARwDO[eY11005_GeneralTowerLightInd_Yellow].00,
    bTowerLightGREEN => ARwDO[eY11006_GeneralTowerLightInd_Green].00); // fbTowerLightCtrl
ARwDO[eY11004_GeneralTowerLightInd_Red].00 := TLctrl.bTowerLightRED;

// NETWORK 2
CLKPLS(bCpStart := TRUE, INT_TIME_ms := 1000); // CLOCK_PLS
CP := CLKPLS.CLOCK_PLS_BOOL;

// NETWORK 3
bAlarmOccurFlagIND := bAlarmOccurFlag AND CP;

// NETWORK 4
//   ARwDO[eY11000_GeneralAlarmResetInd].00: GENERAL ALARM RESET IND (-100S1)
ARwDO[eY11000_GeneralAlarmResetInd].00 := bAlarmOccurFlagIND;

// NETWORK 5
bBuzzerFlagIND := ARbDO[eY11002_GENERALBUZZERTONE01] AND CP;

// NETWORK 6
//   ARwDO[eY11001_GeneralBuzzerResetInd].00: GENERAL BUZZER RESET IND (-100S2)
ARwDO[eY11001_GeneralBuzzerResetInd].00 := bBuzzerFlagIND;

// NETWORK 7
PowerOnDelay(IN := bDCPowerModeActivated AND bIndusoftStart OR ManualPageEnable AND NOT bIndusoftStart OR TRUE, PT := t#10s); // TON

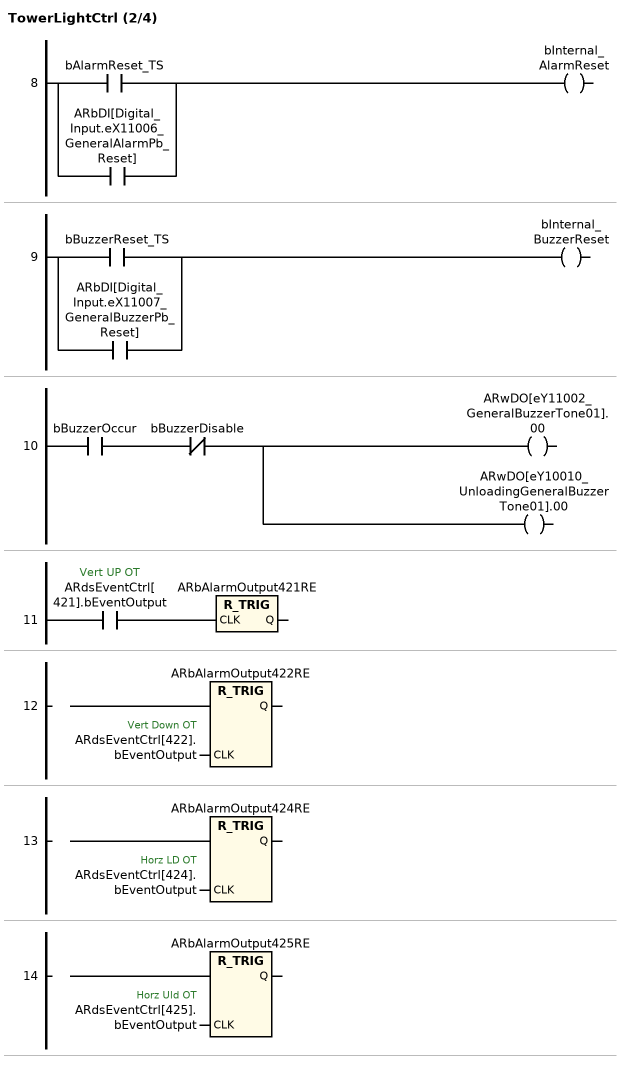
// NETWORK 8
bInternal_AlarmReset := bAlarmReset_TS OR ARbDI[Digital_Input.eX11006_GeneralAlarmPb_Reset];

// NETWORK 9
bInternal_BuzzerReset := bBuzzerReset_TS OR ARbDI[Digital_Input.eX11007_GeneralBuzzerPb_Reset];

// NETWORK 10
_w1 := bBuzzerOccur AND NOT bBuzzerDisable;
ARwDO[eY11002_GeneralBuzzerTone01].00 := _w1;
ARwDO[eY10010_UnloadingGeneralBuzzerTone01].00 := _w1;

// NETWORK 11
//   ARdsEventCtrl[421].bEventOutput: Vert UP OT
ARbAlarmOutput421RE(CLK := ARdsEventCtrl[421].bEventOutput); // R_TRIG

// NETWORK 12
//   ARdsEventCtrl[422].bEventOutput: Vert Down OT
ARbAlarmOutput422RE(CLK := ARdsEventCtrl[422].bEventOutput); // R_TRIG

// NETWORK 13
//   ARdsEventCtrl[424].bEventOutput: Horz LD OT
ARbAlarmOutput424RE(CLK := ARdsEventCtrl[424].bEventOutput); // R_TRIG

// NETWORK 14
//   ARdsEventCtrl[425].bEventOutput: Horz Uld OT
ARbAlarmOutput425RE(CLK := ARdsEventCtrl[425].bEventOutput); // R_TRIG

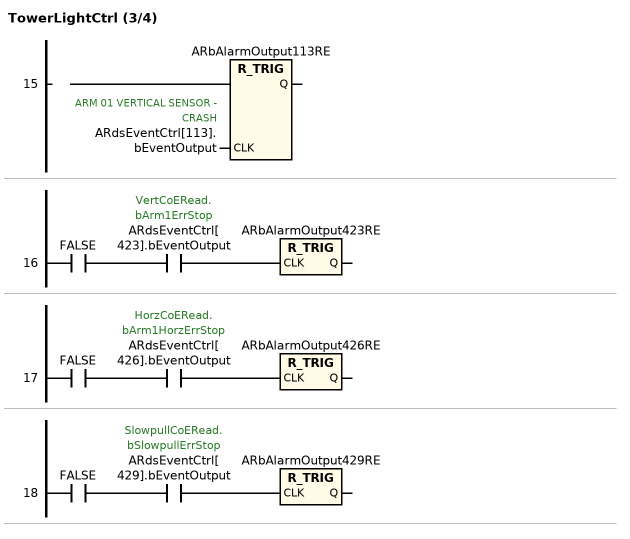
// NETWORK 15
//   ARdsEventCtrl[113].bEventOutput: ARM 01 VERTICAL SENSOR - CRASH
ARbAlarmOutput113RE(CLK := ARdsEventCtrl[113].bEventOutput); // R_TRIG

// NETWORK 16
//   ARdsEventCtrl[423].bEventOutput: VertCoERead.bArm1ErrStop
ARbAlarmOutput423RE(CLK := FALSE AND ARdsEventCtrl[423].bEventOutput); // R_TRIG

// NETWORK 17
//   ARdsEventCtrl[426].bEventOutput: HorzCoERead.bArm1HorzErrStop
ARbAlarmOutput426RE(CLK := FALSE AND ARdsEventCtrl[426].bEventOutput); // R_TRIG

// NETWORK 18
//   ARdsEventCtrl[429].bEventOutput: SlowpullCoERead.bSlowpullErrStop
ARbAlarmOutput429RE(CLK := FALSE AND ARdsEventCtrl[429].bEventOutput); // R_TRIG

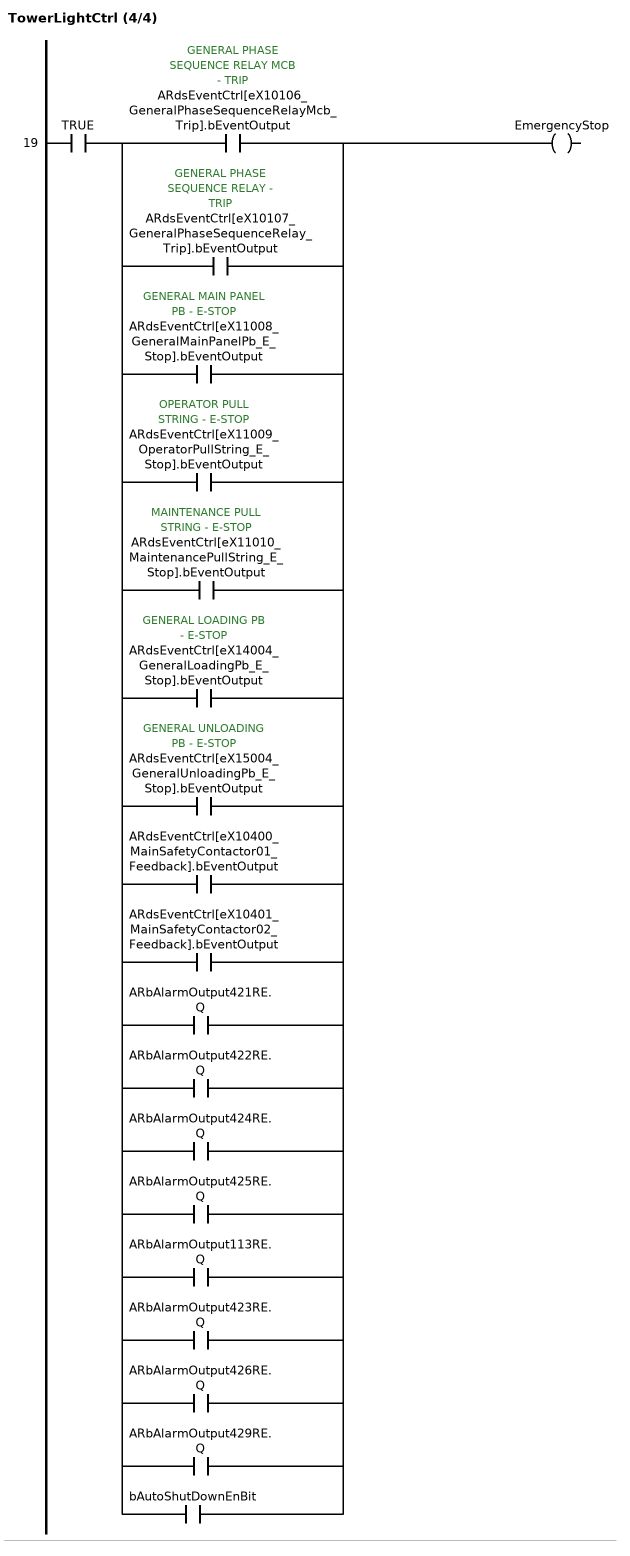
// NETWORK 19
//   ARdsEventCtrl[eX10106_GeneralPhaseSequenceRelayMcb_Trip].bEventOutput: GENERAL PHASE SEQUENCE RELAY MCB - TRIP
//   ARdsEventCtrl[eX10107_GeneralPhaseSequenceRelay_Trip].bEventOutput: GENERAL PHASE SEQUENCE RELAY - TRIP
//   ARdsEventCtrl[eX11008_GeneralMainPanelPb_E_Stop].bEventOutput: GENERAL MAIN PANEL PB - E-STOP
//   ARdsEventCtrl[eX11009_OperatorPullString_E_Stop].bEventOutput: OPERATOR PULL STRING - E-STOP
//   ARdsEventCtrl[eX11010_MaintenancePullString_E_Stop].bEventOutput: MAINTENANCE PULL STRING - E-STOP
//   ARdsEventCtrl[eX14004_GeneralLoadingPb_E_Stop].bEventOutput: GENERAL LOADING PB - E-STOP
//   ARdsEventCtrl[eX15004_GeneralUnloadingPb_E_Stop].bEventOutput: GENERAL UNLOADING PB - E-STOP
EmergencyStop := TRUE AND (ARdsEventCtrl[eX10106_GeneralPhaseSequenceRelayMcb_Trip].bEventOutput OR ARdsEventCtrl[eX10107_GeneralPhaseSequenceRelay_Trip].bEventOutput OR ARdsEventCtrl[eX11008_GeneralMainPanelPb_E_Stop].bEventOutput OR ARdsEventCtrl[eX11009_OperatorPullString_E_Stop].bEventOutput OR ARdsEventCtrl[eX11010_MaintenancePullString_E_Stop].bEventOutput OR ARdsEventCtrl[eX14004_GeneralLoadingPb_E_Stop].bEventOutput OR ARdsEventCtrl[eX15004_GeneralUnloadingPb_E_Stop].bEventOutput OR ARdsEventCtrl[eX10400_MainSafetyContactor01_Feedback].bEventOutput OR ARdsEventCtrl[eX10401_MainSafetyContactor02_Feedback].bEventOutput OR ARbAlarmOutput421RE.Q OR ARbAlarmOutput422RE.Q OR ARbAlarmOutput424RE.Q OR ARbAlarmOutput425RE.Q OR ARbAlarmOutput113RE.Q OR ARbAlarmOutput423RE.Q OR ARbAlarmOutput426RE.Q OR ARbAlarmOutput429RE.Q OR bAutoShutDownEnBit);

END_PROGRAM

// ---- FBs/B_JKS_NewFB/FBP-TowerLightCtrl/fbTowerLightCtrl.TcPOU
FUNCTION_BLOCK fbTowerLightCtrl
VAR_INPUT

	bAlarmOccur : BOOL;
	bMainOnOff : BOOL;
	bAutoPreparationStart : BOOL;
	bAutoPreparationCompleted : BOOL;
	bAutoOriginStart : BOOL;
	bAutoOriginCompleted : BOOL;
	bAutoStart : BOOL;
	bAutoProgress : BOOL;
	bAutoCycleStop: BOOL;
	bManualMode : BOOL;



END_VAR
VAR_OUTPUT
	bTowerLightRED : BOOL;
	bTowerLightYELLOW : BOOL;
	bTowerLightGREEN : BOOL;

END_VAR
VAR

	AlwaysOn : BOOL := TRUE;

	T1: TON;
	T2: TON;
END_VAR

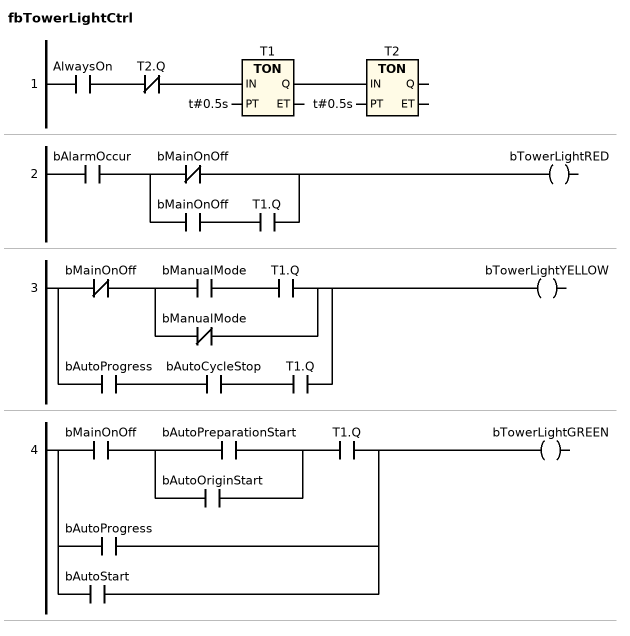
// NETWORK 1
T1(IN := AlwaysOn AND NOT T2.Q, PT := t#0.5s); // TON
T2(IN := T1.Q, PT := t#0.5s); // TON

// NETWORK 2
bTowerLightRED := bAlarmOccur AND (NOT bMainOnOff OR bMainOnOff AND T1.Q);

// NETWORK 3
bTowerLightYELLOW := NOT bMainOnOff AND (bManualMode AND T1.Q OR NOT bManualMode) OR bAutoProgress AND bAutoCycleStop AND T1.Q;

// NETWORK 4
bTowerLightGREEN := (bMainOnOff AND (bAutoPreparationStart OR bAutoOriginStart)) AND T1.Q OR bAutoProgress OR bAutoStart;

END_FUNCTION_BLOCK

// ---- FBs/B_JKS_OldFB/Timer/CLOCK_PLS.TcPOU
FUNCTION_BLOCK CLOCK_PLS
VAR_INPUT
	bCpStart			: BOOL;
	INT_TIME_ms 	: INT;

END_VAR
VAR_OUTPUT
	CLOCK_PLS_BOOL: BOOL;
END_VAR
VAR
	T0: TON;
	T1: TON;
	M0: BOOL;
	M1: BOOL;
	D0: TIME;
	D1: TIME;
END_VAR

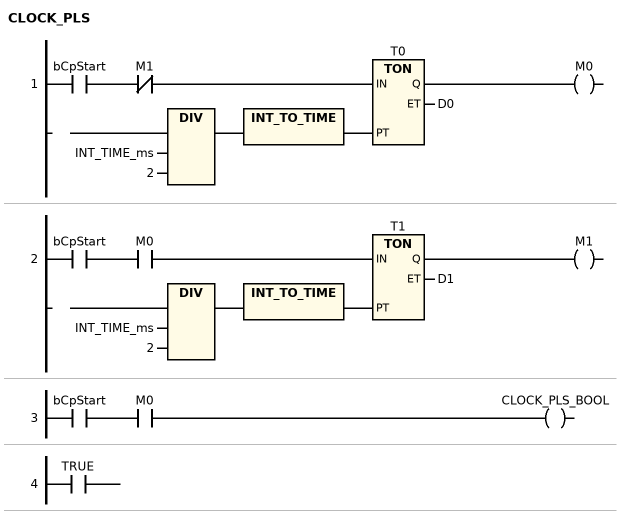
// NETWORK 1
T0(IN := bCpStart AND NOT M1, PT := INT_TO_TIME(INT_TIME_ms / 2), ET => D0); // TON
M0 := T0.Q;

// NETWORK 2
T1(IN := bCpStart AND M0, PT := INT_TO_TIME(INT_TIME_ms / 2), ET => D1); // TON
M1 := T1.Q;

// NETWORK 3
CLOCK_PLS_BOOL := bCpStart AND M0;

// NETWORK 4

END_FUNCTION_BLOCK

// ---- POUs/MainProgram/User/UserCtrl.TcPOU
PROGRAM UserCtrl
VAR

FECloseLoginPage: F_TRIG;

	
	bUserLoginOnPB: BOOL;
END_VAR


// User Group List.. To match with JKS standard
//sUserGroupName[0]			:= 	STRING_TO_WSTRING('');
sUserGroupName[1]			:= 	STRING_TO_WSTRING('OPERATOR');
sUserGroupName[2]			:=	STRING_TO_WSTRING('TECHNICIAN');
sUserGroupName[3]			:=	STRING_TO_WSTRING('ENGINEER');
sUserGroupName[4]			:=	STRING_TO_WSTRING('ADMIN');
//sUserGroupName[5]			:=	STRING_TO_WSTRING('');
//sUserGroupName[6]			:=	STRING_TO_WSTRING('');
//sUserGroupName[7]			:=	STRING_TO_WSTRING('');	

bUserGroupPageON;



// User Ctrl FB
fbHmiTF1800_UserlevelManagement(
	bLoginPB						:= bLoginPB, 
	bLogoutPB						:= bLogoutPB, 
	iLoginNameId					:= iLoginNameId, 
	sPasswordField					:= sPasswordField, 
	iUM_SelectedLoginNameId			:= iUM_SelectedLoginNameId, 
	sUM_CurrentPassword				:= sUM_CurrentPassword, 
	sUM_NewPassword					:= sUM_NewPassword, 
	sUM_ConfirmPassword				:= sUM_ConfirmPassword, 
	sUM_NewUserLoginName			:= sUM_NewUserLoginName, 
	sUM_NewUserGroupId				:= sUM_NewUserGroupId, 
	sUM_NewUserOperatorIdentifier	:= sUM_NewUserOperatorIdentifier, 
	sUM_NewUserActorType			:= sUM_NewUserActorType, 
	sUM_NewUserLastName				:= sUM_NewUserLastName, 
	sUM_NewUserFirstName			:= sUM_NewUserFirstName, 
	bUM_CreatePB					:= bUM_CreatePB, 
	bUM_EditPB						:= bUM_EditPB, 
	bUM_DeletePB					:= bUM_DeletePB, 
	bUM_EnablePB					:= bUM_EnablePB, 
	bUM_DisablePB					:= bUM_DisablePB, 
	bUM_ConfirmPB					:= bUM_ConfirmPB, 
	bUM_ReturnPB					:= bUM_ReturnPB,  
	dsHmiUserStatus_Active			=> dsHmiUserStatus_Active, 
	dsHmiUserStatus_Login			=> dsHmiUserStatus_Login, 
	dsHmiUserStatus_Logout			=> dsHmiUserStatus_Logout, 
	wsActiveUserGroupName			=> sActiveUserGroupname,//VisuElems.CurrentUserName, 						//**, 
	sMessage						=> sMessage);

//Auto switch off the PB (* TESTING USED ONLY)
IF bLoginPB 		THEN	bLoginPB 		:= FALSE;	END_IF
IF bLogoutPB 		THEN	bLogoutPB 		:= FALSE;	END_IF
IF bUM_CreatePB 	THEN	bUM_CreatePB 	:= FALSE;	END_IF
IF bUM_EditPB 		THEN	bUM_EditPB 		:= FALSE;	END_IF
IF bUM_DeletePB 	THEN	bUM_DeletePB 	:= FALSE;	END_IF
IF bUM_EnablePB 	THEN	bUM_EnablePB 	:= FALSE;	END_IF
IF bUM_DisablePB 	THEN	bUM_DisablePB 	:= FALSE;	END_IF
IF bUM_ConfirmPB 	THEN	bUM_ConfirmPB 	:= FALSE;	END_IF
IF bUM_ReturnPB 	THEN	bUM_ReturnPB 	:= FALSE;	END_IF

//HMI CTRL
FECloseLoginPage(CLK:=fbHmiTF1800_UserlevelManagement.dsHmiUserStatus_Login.bActivatedFlag , Q=> );

iCurrentUserGroupID :=fbHmiTF1800_UserlevelManagement.dsHmiUserStatus_Active.sUserGroupId;
//Login Page auto close after user login
IF FECloseLoginPage.Q THEN
	VisuElems.CURRENTVISU := 'AutoMain_Page';
END_IF

//IF 	bUserPageCreateON THEN
//	bUserPageEditON:= FALSE;
//END_IF
		
// Password Field
IF sUM_CurrentPassword<>'' THEN
	sCurrentPwField := '****';
	ELSE
	sCurrentPwField := '';
END_IF

IF sUM_ConfirmPassword<>'' THEN
	sConfirmPwField := '****';
	ELSE
	sConfirmPwField := '';
END_IF

IF sUM_NewPassword<>'' THEN
	sNewPwField := '****';
	ELSE
	sNewPwField := '';
END_IF		

IF sPasswordField<>'' THEN
	sPwField := '****';
	ELSE
	sPwField := '';
END_IF	


iLoginNameId;
sPasswordField;

iUM_SelectedLoginNameId;
fbHmiTF1800_UserlevelManagement.dsHmiUserStatus_Active.sLoginName; //current username

fbHmiTF1800_UserlevelManagement.dsHmiUserStatus_Login.bActivatedFlag;
fbHmiTF1800_UserlevelManagement.dsHmiUserReg.ARwsUserGroupName[iUM_SelectedLoginNameId];
sUM_NewUserActorType;
fbHmiTF1800_UserlevelManagement;
	
//dsHmiUserStatus_Active.bActivatedFlag	;//	:= dsHmiUserStatus_Active.bActivatedFlag; 
//dsHmiUserStatus_Active.eActorType		;//	:= dsHmiUserStatus_Active.sActorType;
//dsHmiUserStatus_Active.sFirstName		;//	:= dsHmiUserStatus_Active.sFirstName; 
//dsHmiUserStatus_Active.sLoginName		;//	:= dsHmiUserStatus_Active.sLoginName; 
//dsHmiUserStatus_Active.sOperatorIdentifier	;//:= dsHmiUserStatus_Active.sOperatorIdentifier; 
//dsHmiUserStatus_Active.sULastName		;//	:= dsHmiUserStatus_Active.sULastName; 
//dsHmiUserStatus_Active.sUserGroupId		;//	:= VisuElems.CurrentUserGroupId; 			//** 	
//dsHmiUserStatus_Active.tsDateTime.wYear;
//dsHmiUserStatus_Active.tsDateTime.wMonth;
//dsHmiUserStatus_Active.tsDateTime.wDay;

//dsHmiUserStatus_Login.bActivatedFlag		;
//dsHmiUserStatus_Login.eActorType			;
//dsHmiUserStatus_Login.sFirstName			;
//dsHmiUserStatus_Login.sLoginName			;
//dsHmiUserStatus_Login.sOperatorIdentifier	;
//dsHmiUserStatus_Login.sULastName			;
//dsHmiUserStatus_Login.sUserGroupId			;
//dsHmiUserStatus_Login.tsDateTime.wYear;
//dsHmiUserStatus_Login.tsDateTime.wMonth;
//dsHmiUserStatus_Login.tsDateTime.wDay;
//dsHmiUserStatus_Login.tsDateTime.wHour;
//dsHmiUserStatus_Login.tsDateTime.wMinute;
//dsHmiUserStatus_Login.tsDateTime.wSecond;
//dsHmiUserStatus_Login.tsDateTime.wMilliseconds;
//dsHmiUserStatus_Login.tsDateTime.wDayOfWeek;
	
//dsHmiUserStatus_Logout.bActivatedFlag		;
//dsHmiUserStatus_Logout.eActorType			;
//dsHmiUserStatus_Logout.sFirstName			;
//dsHmiUserStatus_Logout.sLoginName			;
//dsHmiUserStatus_Logout.sOperatorIdentifier	;
//dsHmiUserStatus_Logout.sULastName			;
//dsHmiUserStatus_Logout.sUserGroupId			;
//dsHmiUserStatus_Logout.tsDateTime.wYear;
//dsHmiUserStatus_Logout.tsDateTime.wMonth;
//dsHmiUserStatus_Logout.tsDateTime.wDay;


//FBCreateGUID(
//	bExecute:= bTestStart, 
//	sNetId:= '', 
//	tTimeout:= T#1S, 
//	pGuidBuffer:= ADR(guGUIDTest), 
//	nGuidBufferSize:= SIZEOF(guGUIDTest), 
//	bBusy=>, 
//	bError=> , 
//	nErrorId=> );
	
//FBCreateGUID.bBusy;
//FBCreateGUID.bError;
//FBCreateGUID.nErrorId;
	
////guGUIDTest := regstring_to_guid(fbHmiTF1800_UserlevelManagement.dsHmiUserReg.ARsPw[1]);
//sGuidOutput := guid_to_regstring(guGUIDTest);
//sGuidOutput2 := guid_to_string(guGUIDTest);
	
	fbHmiTF1800_UserlevelManagement.dsHmiUserReg.ARbUserStatus[1];
	fbHmiTF1800_UserlevelManagement.dsHmiUserReg.AReActorType[1];
	fbHmiTF1800_UserlevelManagement.dsHmiUserReg.ARiUserGroupID[1];
	fbHmiTF1800_UserlevelManagement.dsHmiUserReg.ARsFirstName[1];
	fbHmiTF1800_UserlevelManagement.dsHmiUserReg.ARsLastName[1];
	fbHmiTF1800_UserlevelManagement.dsHmiUserReg.ARsLoginName[1];
	fbHmiTF1800_UserlevelManagement.dsHmiUserReg.ARsOperatorIdentifier[1];
	fbHmiTF1800_UserlevelManagement.dsHmiUserReg.ARsPw[1];
	fbHmiTF1800_UserlevelManagement.dsHmiUserReg.ARwsUserGroupName[1];
	fbHmiTF1800_UserlevelManagement.dsHmiUserReg.iQtyUserReg;
//	fbHmiTF1800_UserlevelManagement.dsHmiUserReg
//	fbHmiTF1800_UserlevelManagement.dsHmiUserReg
//	fbHmiTF1800_UserlevelManagement.dsHmiUserReg
//	fbHmiTF1800_UserlevelManagement.dsHmiUserReg
//	fbHmiTF1800_UserlevelManagement.dsHmiUserReg


	fbHmiTF1800_UserlevelManagement.dsHmiUserReg.ARbUserStatus[iUM_SelectedLoginNameId];
	fbHmiTF1800_UserlevelManagement.dsHmiUserReg.AReActorType[iUM_SelectedLoginNameId];
	fbHmiTF1800_UserlevelManagement.dsHmiUserReg.ARiUserGroupID[iUM_SelectedLoginNameId];
	fbHmiTF1800_UserlevelManagement.dsHmiUserReg.ARsFirstName[iUM_SelectedLoginNameId];
	fbHmiTF1800_UserlevelManagement.dsHmiUserReg.ARsLastName[iUM_SelectedLoginNameId];
	fbHmiTF1800_UserlevelManagement.dsHmiUserReg.ARsLoginName[iUM_SelectedLoginNameId];
	fbHmiTF1800_UserlevelManagement.dsHmiUserReg.ARsOperatorIdentifier[iUM_SelectedLoginNameId];
	fbHmiTF1800_UserlevelManagement.dsHmiUserReg.ARsPw[iUM_SelectedLoginNameId];
	fbHmiTF1800_UserlevelManagement.dsHmiUserReg.ARwsUserGroupName[iUM_SelectedLoginNameId];
	fbHmiTF1800_UserlevelManagement.dsHmiUserReg.ARwsUserGroupName[iUM_SelectedLoginNameId];

	
	fbHmiTF1800_UserlevelManagement.dsHmiUserReg.ARbUserStatus[2];
	fbHmiTF1800_UserlevelManagement.dsHmiUserReg.AReActorType[2];
	fbHmiTF1800_UserlevelManagement.dsHmiUserReg.ARiUserGroupID[2];
	fbHmiTF1800_UserlevelManagement.dsHmiUserReg.ARsFirstName[2];
	fbHmiTF1800_UserlevelManagement.dsHmiUserReg.ARsLastName[2];
	fbHmiTF1800_UserlevelManagement.dsHmiUserReg.ARsLoginName[2];
	fbHmiTF1800_UserlevelManagement.dsHmiUserReg.ARsOperatorIdentifier[2];
	fbHmiTF1800_UserlevelManagement.dsHmiUserReg.ARsPw[2];
	fbHmiTF1800_UserlevelManagement.dsHmiUserReg.ARwsUserGroupName[2];
//	fbHmiTF1800_UserlevelManagement.dsHmiUserReg.iQtyUserReg[2];

	fbHmiTF1800_UserlevelManagement.dsHmiUserReg.ARbUserStatus[3];
	fbHmiTF1800_UserlevelManagement.dsHmiUserReg.AReActorType[3];
	fbHmiTF1800_UserlevelManagement.dsHmiUserReg.ARiUserGroupID[3];
	fbHmiTF1800_UserlevelManagement.dsHmiUserReg.ARsFirstName[3];
	fbHmiTF1800_UserlevelManagement.dsHmiUserReg.ARsLastName[3];
	fbHmiTF1800_UserlevelManagement.dsHmiUserReg.ARsLoginName[3];
	fbHmiTF1800_UserlevelManagement.dsHmiUserReg.ARsOperatorIdentifier[3];
	fbHmiTF1800_UserlevelManagement.dsHmiUserReg.ARsPw[3];
	fbHmiTF1800_UserlevelManagement.dsHmiUserReg.ARwsUserGroupName[3];
//	fbHmiTF1800_UserlevelManagement.dsHmiUserReg.iQtyUserReg[3];	
	
	
	fbHmiTF1800_UserlevelManagement.dsHmiUserReg.ARbUserStatus[4];
	fbHmiTF1800_UserlevelManagement.dsHmiUserReg.AReActorType[4];
	fbHmiTF1800_UserlevelManagement.dsHmiUserReg.ARiUserGroupID[4];
	fbHmiTF1800_UserlevelManagement.dsHmiUserReg.ARsFirstName[4];
	fbHmiTF1800_UserlevelManagement.dsHmiUserReg.ARsLastName[4];
	fbHmiTF1800_UserlevelManagement.dsHmiUserReg.ARsLoginName[4];
	fbHmiTF1800_UserlevelManagement.dsHmiUserReg.ARsOperatorIdentifier[4];
	fbHmiTF1800_UserlevelManagement.dsHmiUserReg.ARsPw[4];
	fbHmiTF1800_UserlevelManagement.dsHmiUserReg.ARwsUserGroupName[4];
//	fbHmiTF1800_UserlevelManagement.dsHmiUserReg.iQtyUserReg[4];	
	
	fbHmiTF1800_UserlevelManagement.dsHmiUserReg.ARbUserStatus[5];
	fbHmiTF1800_UserlevelManagement.dsHmiUserReg.AReActorType[5];
	fbHmiTF1800_UserlevelManagement.dsHmiUserReg.ARiUserGroupID[5];
	fbHmiTF1800_UserlevelManagement.dsHmiUserReg.ARsFirstName[5];
	fbHmiTF1800_UserlevelManagement.dsHmiUserReg.ARsLastName[5];
	fbHmiTF1800_UserlevelManagement.dsHmiUserReg.ARsLoginName[5];
	fbHmiTF1800_UserlevelManagement.dsHmiUserReg.ARsOperatorIdentifier[5];
	fbHmiTF1800_UserlevelManagement.dsHmiUserReg.ARsPw[5];
	fbHmiTF1800_UserlevelManagement.dsHmiUserReg.ARwsUserGroupName[5];
//	fbHmiTF1800_UserlevelManagement.dsHmiUserReg.iQtyUserReg[5];

	fbHmiTF1800_UserlevelManagement.dsHmiUserReg.ARbUserStatus[6];
	fbHmiTF1800_UserlevelManagement.dsHmiUserReg.AReActorType[6];
	fbHmiTF1800_UserlevelManagement.dsHmiUserReg.ARiUserGroupID[6];
	fbHmiTF1800_UserlevelManagement.dsHmiUserReg.ARsFirstName[6];
	fbHmiTF1800_UserlevelManagement.dsHmiUserReg.ARsLastName[6];
	fbHmiTF1800_UserlevelManagement.dsHmiUserReg.ARsLoginName[6];
	fbHmiTF1800_UserlevelManagement.dsHmiUserReg.ARsOperatorIdentifier[6];
	fbHmiTF1800_UserlevelManagement.dsHmiUserReg.ARsPw[6];
	fbHmiTF1800_UserlevelManagement.dsHmiUserReg.ARwsUserGroupName[6];
//	fbHmiTF1800_UserlevelManagement.dsHmiUserReg.iQtyUserReg[6];
	
	fbHmiTF1800_UserlevelManagement.dsHmiUserReg.ARbUserStatus[7];
	fbHmiTF1800_UserlevelManagement.dsHmiUserReg.AReActorType[7];
	fbHmiTF1800_UserlevelManagement.dsHmiUserReg.ARiUserGroupID[7];
	fbHmiTF1800_UserlevelManagement.dsHmiUserReg.ARsFirstName[7];
	fbHmiTF1800_UserlevelManagement.dsHmiUserReg.ARsLastName[7];
	fbHmiTF1800_UserlevelManagement.dsHmiUserReg.ARsLoginName[7];
	fbHmiTF1800_UserlevelManagement.dsHmiUserReg.ARsOperatorIdentifier[7];
	fbHmiTF1800_UserlevelManagement.dsHmiUserReg.ARsPw[7];
	fbHmiTF1800_UserlevelManagement.dsHmiUserReg.ARwsUserGroupName[7];
//	fbHmiTF1800_UserlevelManagement.dsHmiUserReg.iQtyUserReg[7];	

	fbHmiTF1800_UserlevelManagement.dsHmiUserReg.ARbUserStatus[8];
	fbHmiTF1800_UserlevelManagement.dsHmiUserReg.AReActorType[8];
	fbHmiTF1800_UserlevelManagement.dsHmiUserReg.ARiUserGroupID[8];
	fbHmiTF1800_UserlevelManagement.dsHmiUserReg.ARsFirstName[8];
	fbHmiTF1800_UserlevelManagement.dsHmiUserReg.ARsLastName[8];
	fbHmiTF1800_UserlevelManagement.dsHmiUserReg.ARsLoginName[8];
	fbHmiTF1800_UserlevelManagement.dsHmiUserReg.ARsOperatorIdentifier[8];
	fbHmiTF1800_UserlevelManagement.dsHmiUserReg.ARsPw[8];
	fbHmiTF1800_UserlevelManagement.dsHmiUserReg.ARwsUserGroupName[8];
//	fbHmiTF1800_UserlevelManagement.dsHmiUserReg.iQtyUserReg[8];	
	
	fbHmiTF1800_UserlevelManagement.dsHmiUserReg.ARbUserStatus[9];
	fbHmiTF1800_UserlevelManagement.dsHmiUserReg.AReActorType[9];
	fbHmiTF1800_UserlevelManagement.dsHmiUserReg.ARiUserGroupID[9];
	fbHmiTF1800_UserlevelManagement.dsHmiUserReg.ARsFirstName[9];
	fbHmiTF1800_UserlevelManagement.dsHmiUserReg.ARsLastName[9];
	fbHmiTF1800_UserlevelManagement.dsHmiUserReg.ARsLoginName[9];
	fbHmiTF1800_UserlevelManagement.dsHmiUserReg.ARsOperatorIdentifier[9];
	fbHmiTF1800_UserlevelManagement.dsHmiUserReg.ARsPw[9];
	fbHmiTF1800_UserlevelManagement.dsHmiUserReg.ARwsUserGroupName[9];
//	fbHmiTF1800_UserlevelManagement.dsHmiUserReg.iQtyUserReg[9];	

//	fbHmiTF1800_UserlevelManagement.dsHmiUserReg.ARbUserStatus[1];
//	fbHmiTF1800_UserlevelManagement.dsHmiUserReg.AReActorType[1];
//	fbHmiTF1800_UserlevelManagement.dsHmiUserReg.ARiUserGroupID[1];
//	fbHmiTF1800_UserlevelManagement.dsHmiUserReg.ARsFirstName[1];
//	fbHmiTF1800_UserlevelManagement.dsHmiUserReg.ARsLastName[1];
//	fbHmiTF1800_UserlevelManagement.dsHmiUserReg.ARsLoginName[1];
//	fbHmiTF1800_UserlevelManagement.dsHmiUserReg.ARsOperatorIdentifier[1];
//	fbHmiTF1800_UserlevelManagement.dsHmiUserReg.ARsPw[1];
//	fbHmiTF1800_UserlevelManagement.dsHmiUserReg.ARwsUserGroupName[1];
//	fbHmiTF1800_UserlevelManagement.dsHmiUserReg.iQtyUserReg[1];

END_PROGRAM

// ---- POUs/MainProgram/BasketMemory_RecipeCtrl/BasketBadCtrl.TcPOU
PROGRAM BasketBadCtrl
VAR
	ARfbStnBadAssignCtrl: ARRAY [1..iStnQty] OF fbAssignBadBstCtrl;
	ARfbArmBadAssignCtrl: ARRAY [1..iArmQty] OF fbAssignBadBstCtrl;
	bGeneralAssignBadBasket: BOOL;

END_VAR

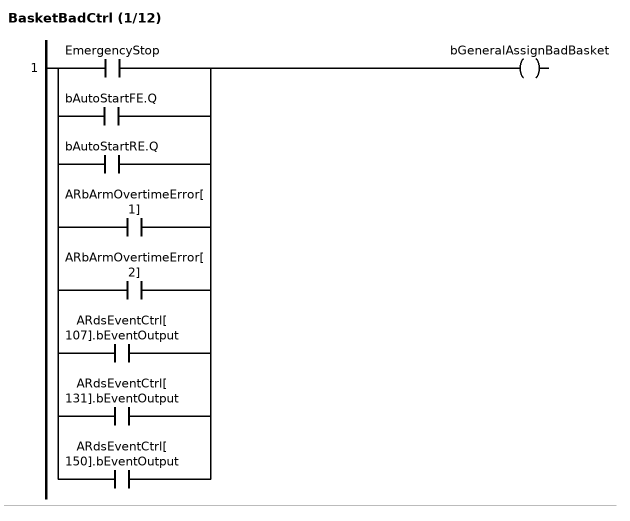
// NETWORK 1
bGeneralAssignBadBasket := EmergencyStop OR bAutoStartFE.Q OR bAutoStartRE.Q OR ARbArmOvertimeError[1] OR ARbArmOvertimeError[2] OR ARdsEventCtrl[107].bEventOutput OR ARdsEventCtrl[131].bEventOutput OR ARdsEventCtrl[150].bEventOutput;

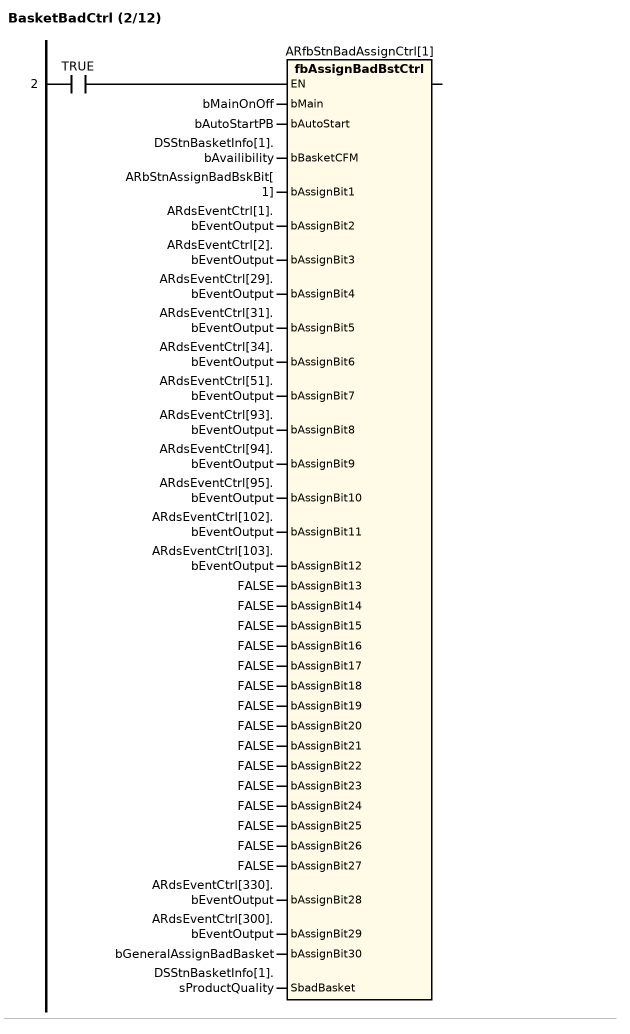
// NETWORK 2
ARfbStnBadAssignCtrl[1](
    bMain := bMainOnOff,
    bAutoStart := bAutoStartPB,
    bBasketCFM := DSStnBasketInfo[1].bAvailibility,
    bAssignBit1 := ARbStnAssignBadBskBit[1],
    bAssignBit2 := ARdsEventCtrl[1].bEventOutput,
    bAssignBit3 := ARdsEventCtrl[2].bEventOutput,
    bAssignBit4 := ARdsEventCtrl[29].bEventOutput,
    bAssignBit5 := ARdsEventCtrl[31].bEventOutput,
    bAssignBit6 := ARdsEventCtrl[34].bEventOutput,
    bAssignBit7 := ARdsEventCtrl[51].bEventOutput,
    bAssignBit8 := ARdsEventCtrl[93].bEventOutput,
    bAssignBit9 := ARdsEventCtrl[94].bEventOutput,
    bAssignBit10 := ARdsEventCtrl[95].bEventOutput,
    bAssignBit11 := ARdsEventCtrl[102].bEventOutput,
    bAssignBit12 := ARdsEventCtrl[103].bEventOutput,
    bAssignBit13 := FALSE,
    bAssignBit14 := FALSE,
    bAssignBit15 := FALSE,
    bAssignBit16 := FALSE,
    bAssignBit17 := FALSE,
    bAssignBit18 := FALSE,
    bAssignBit19 := FALSE,
    bAssignBit20 := FALSE,
    bAssignBit21 := FALSE,
    bAssignBit22 := FALSE,
    bAssignBit23 := FALSE,
    bAssignBit24 := FALSE,
    bAssignBit25 := FALSE,
    bAssignBit26 := FALSE,
    bAssignBit27 := FALSE,
    bAssignBit28 := ARdsEventCtrl[330].bEventOutput,
    bAssignBit29 := ARdsEventCtrl[300].bEventOutput,
    bAssignBit30 := bGeneralAssignBadBasket,
    SbadBasket := DSStnBasketInfo[1].sProductQuality); // fbAssignBadBstCtrl

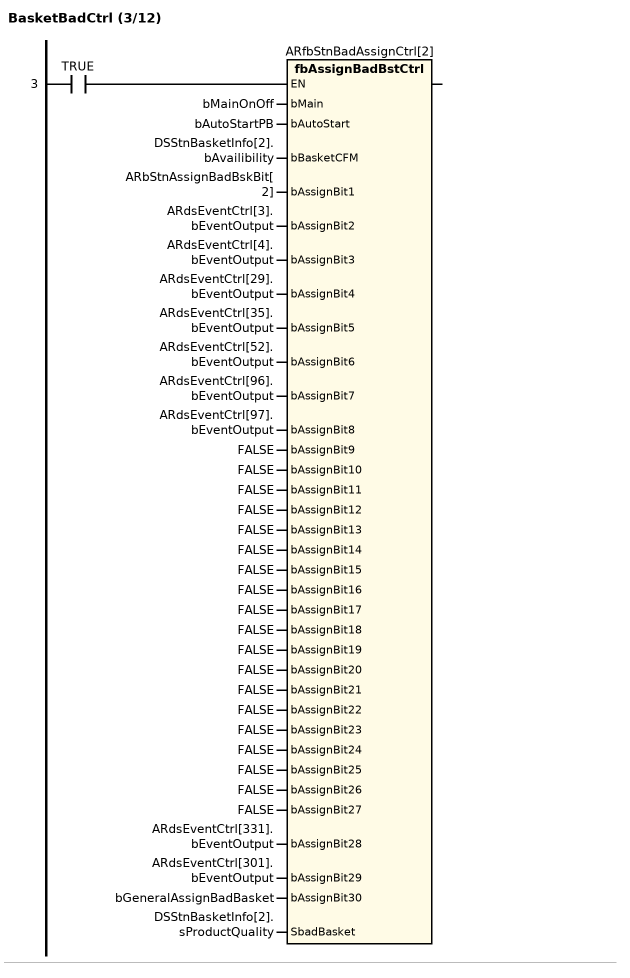
// NETWORK 3
ARfbStnBadAssignCtrl[2](
    bMain := bMainOnOff,
    bAutoStart := bAutoStartPB,
    bBasketCFM := DSStnBasketInfo[2].bAvailibility,
    bAssignBit1 := ARbStnAssignBadBskBit[2],
    bAssignBit2 := ARdsEventCtrl[3].bEventOutput,
    bAssignBit3 := ARdsEventCtrl[4].bEventOutput,
    bAssignBit4 := ARdsEventCtrl[29].bEventOutput,
    bAssignBit5 := ARdsEventCtrl[35].bEventOutput,
    bAssignBit6 := ARdsEventCtrl[52].bEventOutput,
    bAssignBit7 := ARdsEventCtrl[96].bEventOutput,
    bAssignBit8 := ARdsEventCtrl[97].bEventOutput,
    bAssignBit9 := FALSE,
    bAssignBit10 := FALSE,
    bAssignBit11 := FALSE,
    bAssignBit12 := FALSE,
    bAssignBit13 := FALSE,
    bAssignBit14 := FALSE,
    bAssignBit15 := FALSE,
    bAssignBit16 := FALSE,
    bAssignBit17 := FALSE,
    bAssignBit18 := FALSE,
    bAssignBit19 := FALSE,
    bAssignBit20 := FALSE,
    bAssignBit21 := FALSE,
    bAssignBit22 := FALSE,
    bAssignBit23 := FALSE,
    bAssignBit24 := FALSE,
    bAssignBit25 := FALSE,
    bAssignBit26 := FALSE,
    bAssignBit27 := FALSE,
    bAssignBit28 := ARdsEventCtrl[331].bEventOutput,
    bAssignBit29 := ARdsEventCtrl[301].bEventOutput,
    bAssignBit30 := bGeneralAssignBadBasket,
    SbadBasket := DSStnBasketInfo[2].sProductQuality); // fbAssignBadBstCtrl

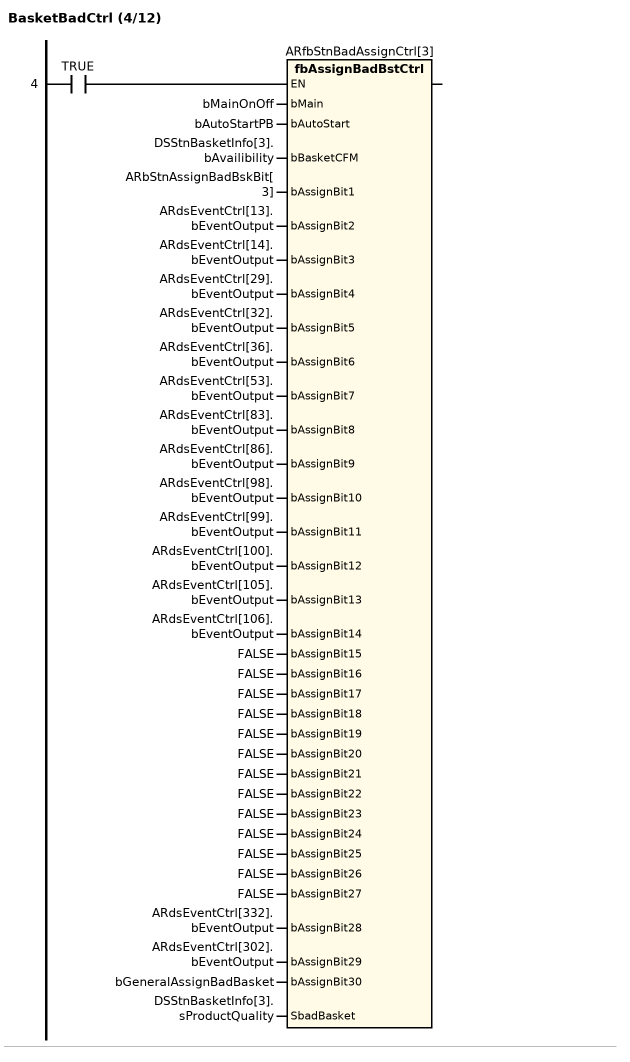
// NETWORK 4
ARfbStnBadAssignCtrl[3](
    bMain := bMainOnOff,
    bAutoStart := bAutoStartPB,
    bBasketCFM := DSStnBasketInfo[3].bAvailibility,
    bAssignBit1 := ARbStnAssignBadBskBit[3],
    bAssignBit2 := ARdsEventCtrl[13].bEventOutput,
    bAssignBit3 := ARdsEventCtrl[14].bEventOutput,
    bAssignBit4 := ARdsEventCtrl[29].bEventOutput,
    bAssignBit5 := ARdsEventCtrl[32].bEventOutput,
    bAssignBit6 := ARdsEventCtrl[36].bEventOutput,
    bAssignBit7 := ARdsEventCtrl[53].bEventOutput,
    bAssignBit8 := ARdsEventCtrl[83].bEventOutput,
    bAssignBit9 := ARdsEventCtrl[86].bEventOutput,
    bAssignBit10 := ARdsEventCtrl[98].bEventOutput,
    bAssignBit11 := ARdsEventCtrl[99].bEventOutput,
    bAssignBit12 := ARdsEventCtrl[100].bEventOutput,
    bAssignBit13 := ARdsEventCtrl[105].bEventOutput,
    bAssignBit14 := ARdsEventCtrl[106].bEventOutput,
    bAssignBit15 := FALSE,
    bAssignBit16 := FALSE,
    bAssignBit17 := FALSE,
    bAssignBit18 := FALSE,
    bAssignBit19 := FALSE,
    bAssignBit20 := FALSE,
    bAssignBit21 := FALSE,
    bAssignBit22 := FALSE,
    bAssignBit23 := FALSE,
    bAssignBit24 := FALSE,
    bAssignBit25 := FALSE,
    bAssignBit26 := FALSE,
    bAssignBit27 := FALSE,
    bAssignBit28 := ARdsEventCtrl[332].bEventOutput,
    bAssignBit29 := ARdsEventCtrl[302].bEventOutput,
    bAssignBit30 := bGeneralAssignBadBasket,
    SbadBasket := DSStnBasketInfo[3].sProductQuality); // fbAssignBadBstCtrl

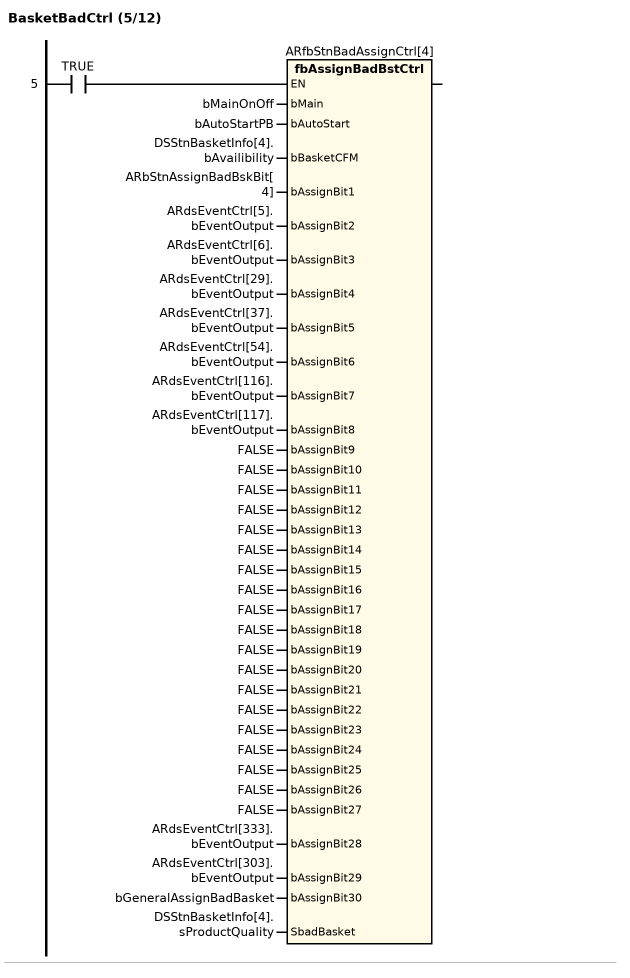
// NETWORK 5
ARfbStnBadAssignCtrl[4](
    bMain := bMainOnOff,
    bAutoStart := bAutoStartPB,
    bBasketCFM := DSStnBasketInfo[4].bAvailibility,
    bAssignBit1 := ARbStnAssignBadBskBit[4],
    bAssignBit2 := ARdsEventCtrl[5].bEventOutput,
    bAssignBit3 := ARdsEventCtrl[6].bEventOutput,
    bAssignBit4 := ARdsEventCtrl[29].bEventOutput,
    bAssignBit5 := ARdsEventCtrl[37].bEventOutput,
    bAssignBit6 := ARdsEventCtrl[54].bEventOutput,
    bAssignBit7 := ARdsEventCtrl[116].bEventOutput,
    bAssignBit8 := ARdsEventCtrl[117].bEventOutput,
    bAssignBit9 := FALSE,
    bAssignBit10 := FALSE,
    bAssignBit11 := FALSE,
    bAssignBit12 := FALSE,
    bAssignBit13 := FALSE,
    bAssignBit14 := FALSE,
    bAssignBit15 := FALSE,
    bAssignBit16 := FALSE,
    bAssignBit17 := FALSE,
    bAssignBit18 := FALSE,
    bAssignBit19 := FALSE,
    bAssignBit20 := FALSE,
    bAssignBit21 := FALSE,
    bAssignBit22 := FALSE,
    bAssignBit23 := FALSE,
    bAssignBit24 := FALSE,
    bAssignBit25 := FALSE,
    bAssignBit26 := FALSE,
    bAssignBit27 := FALSE,
    bAssignBit28 := ARdsEventCtrl[333].bEventOutput,
    bAssignBit29 := ARdsEventCtrl[303].bEventOutput,
    bAssignBit30 := bGeneralAssignBadBasket,
    SbadBasket := DSStnBasketInfo[4].sProductQuality); // fbAssignBadBstCtrl

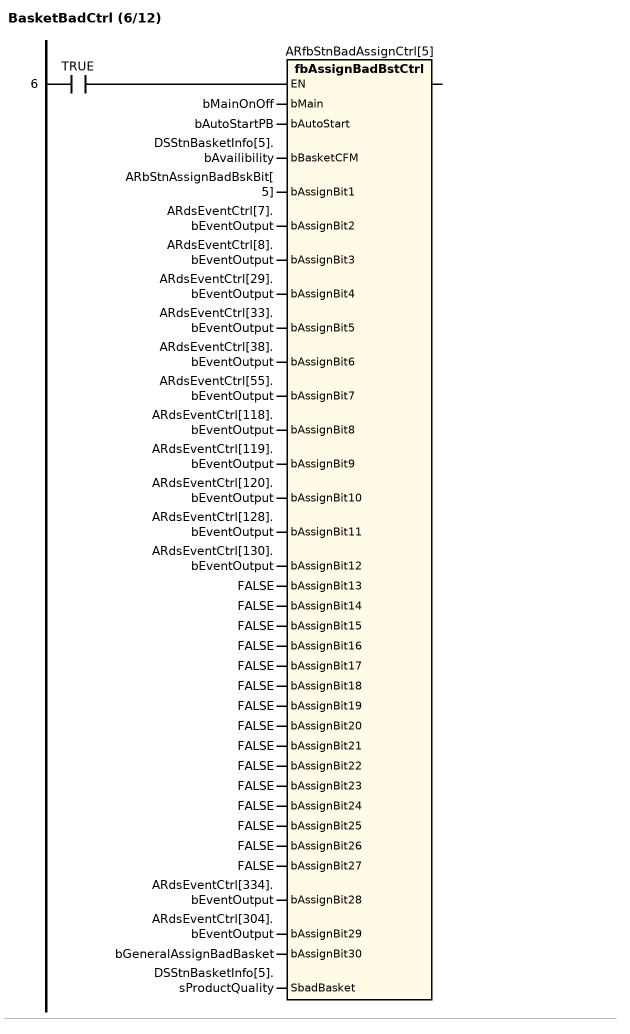
// NETWORK 6
ARfbStnBadAssignCtrl[5](
    bMain := bMainOnOff,
    bAutoStart := bAutoStartPB,
    bBasketCFM := DSStnBasketInfo[5].bAvailibility,
    bAssignBit1 := ARbStnAssignBadBskBit[5],
    bAssignBit2 := ARdsEventCtrl[7].bEventOutput,
    bAssignBit3 := ARdsEventCtrl[8].bEventOutput,
    bAssignBit4 := ARdsEventCtrl[29].bEventOutput,
    bAssignBit5 := ARdsEventCtrl[33].bEventOutput,
    bAssignBit6 := ARdsEventCtrl[38].bEventOutput,
    bAssignBit7 := ARdsEventCtrl[55].bEventOutput,
    bAssignBit8 := ARdsEventCtrl[118].bEventOutput,
    bAssignBit9 := ARdsEventCtrl[119].bEventOutput,
    bAssignBit10 := ARdsEventCtrl[120].bEventOutput,
    bAssignBit11 := ARdsEventCtrl[128].bEventOutput,
    bAssignBit12 := ARdsEventCtrl[130].bEventOutput,
    bAssignBit13 := FALSE,
    bAssignBit14 := FALSE,
    bAssignBit15 := FALSE,
    bAssignBit16 := FALSE,
    bAssignBit17 := FALSE,
    bAssignBit18 := FALSE,
    bAssignBit19 := FALSE,
    bAssignBit20 := FALSE,
    bAssignBit21 := FALSE,
    bAssignBit22 := FALSE,
    bAssignBit23 := FALSE,
    bAssignBit24 := FALSE,
    bAssignBit25 := FALSE,
    bAssignBit26 := FALSE,
    bAssignBit27 := FALSE,
    bAssignBit28 := ARdsEventCtrl[334].bEventOutput,
    bAssignBit29 := ARdsEventCtrl[304].bEventOutput,
    bAssignBit30 := bGeneralAssignBadBasket,
    SbadBasket := DSStnBasketInfo[5].sProductQuality); // fbAssignBadBstCtrl

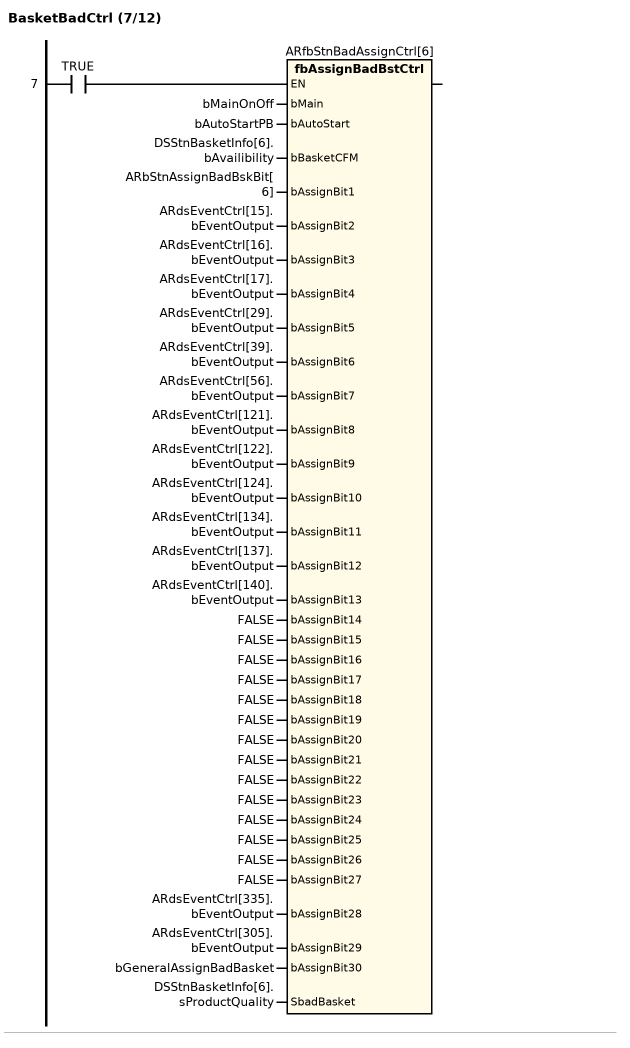
// NETWORK 7
ARfbStnBadAssignCtrl[6](
    bMain := bMainOnOff,
    bAutoStart := bAutoStartPB,
    bBasketCFM := DSStnBasketInfo[6].bAvailibility,
    bAssignBit1 := ARbStnAssignBadBskBit[6],
    bAssignBit2 := ARdsEventCtrl[15].bEventOutput,
    bAssignBit3 := ARdsEventCtrl[16].bEventOutput,
    bAssignBit4 := ARdsEventCtrl[17].bEventOutput,
    bAssignBit5 := ARdsEventCtrl[29].bEventOutput,
    bAssignBit6 := ARdsEventCtrl[39].bEventOutput,
    bAssignBit7 := ARdsEventCtrl[56].bEventOutput,
    bAssignBit8 := ARdsEventCtrl[121].bEventOutput,
    bAssignBit9 := ARdsEventCtrl[122].bEventOutput,
    bAssignBit10 := ARdsEventCtrl[124].bEventOutput,
    bAssignBit11 := ARdsEventCtrl[134].bEventOutput,
    bAssignBit12 := ARdsEventCtrl[137].bEventOutput,
    bAssignBit13 := ARdsEventCtrl[140].bEventOutput,
    bAssignBit14 := FALSE,
    bAssignBit15 := FALSE,
    bAssignBit16 := FALSE,
    bAssignBit17 := FALSE,
    bAssignBit18 := FALSE,
    bAssignBit19 := FALSE,
    bAssignBit20 := FALSE,
    bAssignBit21 := FALSE,
    bAssignBit22 := FALSE,
    bAssignBit23 := FALSE,
    bAssignBit24 := FALSE,
    bAssignBit25 := FALSE,
    bAssignBit26 := FALSE,
    bAssignBit27 := FALSE,
    bAssignBit28 := ARdsEventCtrl[335].bEventOutput,
    bAssignBit29 := ARdsEventCtrl[305].bEventOutput,
    bAssignBit30 := bGeneralAssignBadBasket,
    SbadBasket := DSStnBasketInfo[6].sProductQuality); // fbAssignBadBstCtrl

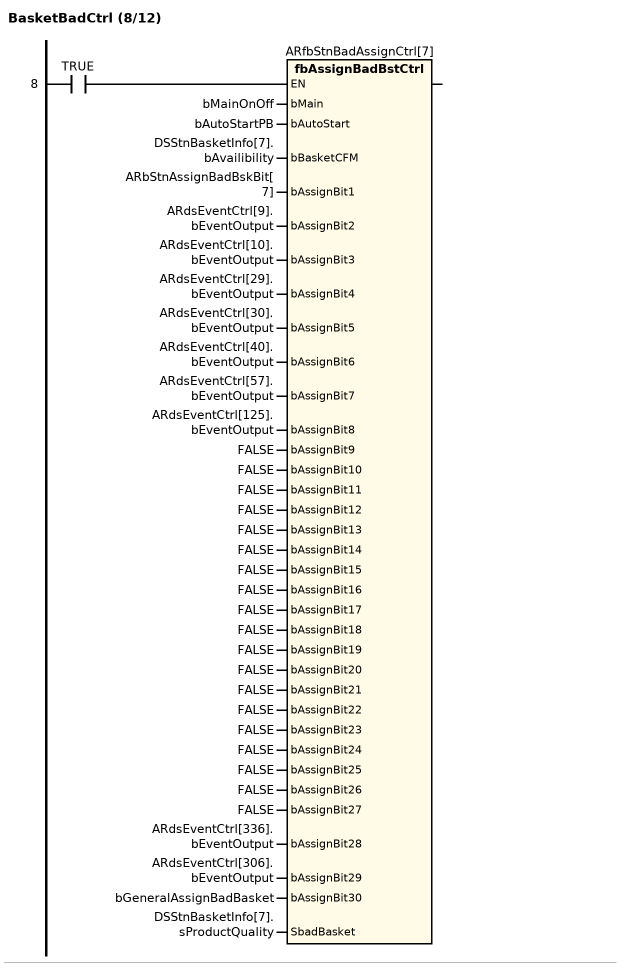
// NETWORK 8
ARfbStnBadAssignCtrl[7](
    bMain := bMainOnOff,
    bAutoStart := bAutoStartPB,
    bBasketCFM := DSStnBasketInfo[7].bAvailibility,
    bAssignBit1 := ARbStnAssignBadBskBit[7],
    bAssignBit2 := ARdsEventCtrl[9].bEventOutput,
    bAssignBit3 := ARdsEventCtrl[10].bEventOutput,
    bAssignBit4 := ARdsEventCtrl[29].bEventOutput,
    bAssignBit5 := ARdsEventCtrl[30].bEventOutput,
    bAssignBit6 := ARdsEventCtrl[40].bEventOutput,
    bAssignBit7 := ARdsEventCtrl[57].bEventOutput,
    bAssignBit8 := ARdsEventCtrl[125].bEventOutput,
    bAssignBit9 := FALSE,
    bAssignBit10 := FALSE,
    bAssignBit11 := FALSE,
    bAssignBit12 := FALSE,
    bAssignBit13 := FALSE,
    bAssignBit14 := FALSE,
    bAssignBit15 := FALSE,
    bAssignBit16 := FALSE,
    bAssignBit17 := FALSE,
    bAssignBit18 := FALSE,
    bAssignBit19 := FALSE,
    bAssignBit20 := FALSE,
    bAssignBit21 := FALSE,
    bAssignBit22 := FALSE,
    bAssignBit23 := FALSE,
    bAssignBit24 := FALSE,
    bAssignBit25 := FALSE,
    bAssignBit26 := FALSE,
    bAssignBit27 := FALSE,
    bAssignBit28 := ARdsEventCtrl[336].bEventOutput,
    bAssignBit29 := ARdsEventCtrl[306].bEventOutput,
    bAssignBit30 := bGeneralAssignBadBasket,
    SbadBasket := DSStnBasketInfo[7].sProductQuality); // fbAssignBadBstCtrl

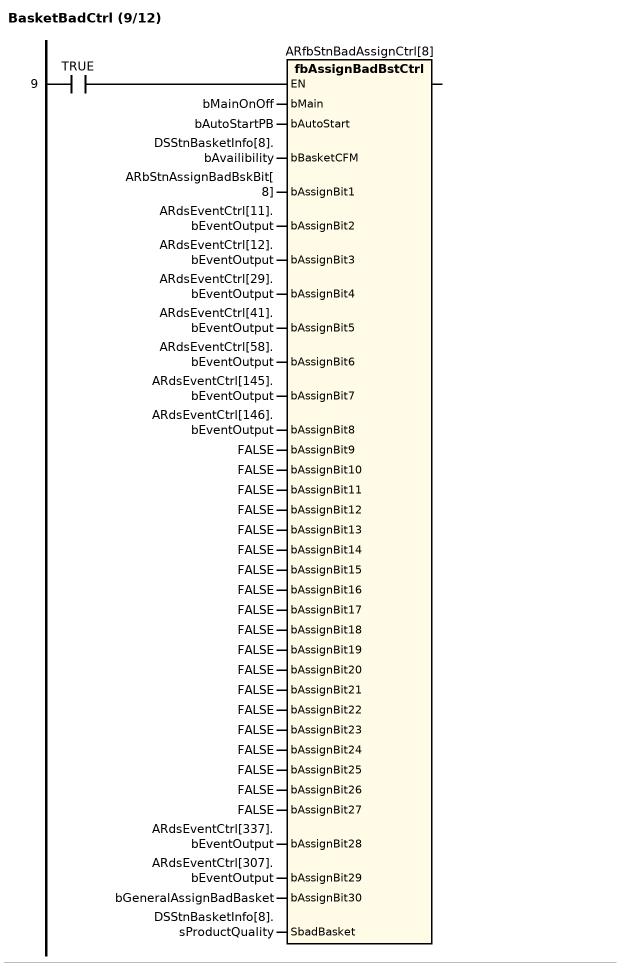
// NETWORK 9
ARfbStnBadAssignCtrl[8](
    bMain := bMainOnOff,
    bAutoStart := bAutoStartPB,
    bBasketCFM := DSStnBasketInfo[8].bAvailibility,
    bAssignBit1 := ARbStnAssignBadBskBit[8],
    bAssignBit2 := ARdsEventCtrl[11].bEventOutput,
    bAssignBit3 := ARdsEventCtrl[12].bEventOutput,
    bAssignBit4 := ARdsEventCtrl[29].bEventOutput,
    bAssignBit5 := ARdsEventCtrl[41].bEventOutput,
    bAssignBit6 := ARdsEventCtrl[58].bEventOutput,
    bAssignBit7 := ARdsEventCtrl[145].bEventOutput,
    bAssignBit8 := ARdsEventCtrl[146].bEventOutput,
    bAssignBit9 := FALSE,
    bAssignBit10 := FALSE,
    bAssignBit11 := FALSE,
    bAssignBit12 := FALSE,
    bAssignBit13 := FALSE,
    bAssignBit14 := FALSE,
    bAssignBit15 := FALSE,
    bAssignBit16 := FALSE,
    bAssignBit17 := FALSE,
    bAssignBit18 := FALSE,
    bAssignBit19 := FALSE,
    bAssignBit20 := FALSE,
    bAssignBit21 := FALSE,
    bAssignBit22 := FALSE,
    bAssignBit23 := FALSE,
    bAssignBit24 := FALSE,
    bAssignBit25 := FALSE,
    bAssignBit26 := FALSE,
    bAssignBit27 := FALSE,
    bAssignBit28 := ARdsEventCtrl[337].bEventOutput,
    bAssignBit29 := ARdsEventCtrl[307].bEventOutput,
    bAssignBit30 := bGeneralAssignBadBasket,
    SbadBasket := DSStnBasketInfo[8].sProductQuality); // fbAssignBadBstCtrl

